CASE nIndex OF
	0: // idle state
		Inspect := 0;
	10: // trigger the camera
		IF GetCameraData() = 1 THEN
			Count := CameraData.Results.Count;
			CountStart := CameraData.Results.Count;
			nIndex := 11;
		END_IF
	11: // trigger camera
		Trigger := TRUE;
		nIndex := 12;
	12: // wait 250 ms
		CameraTON.IN := TRUE;
		IF CameraTON.Q THEN
			CameraTON.IN := FALSE;
			nIndex := 15;
		END_IF
		CameraTON();
	15: // wait for data to be updated
		CameraDataResult := GetCameraData();
		IF CameraDataResult = 1 THEN
			IF Count <> CameraData.Results.Count THEN
				CountFinish := CameraData.Results.Count;
				nIndex := 20;
				Trigger := FALSE;
			END_IF
		END_IF
	20: // Gather the data and analyze locations, etc.
		CameraDataResult := Compute(Execute := TRUE);
		IF CameraDataResult = 1 THEN	// could compute b/c found pattern
			Compute(Execute := FALSE);
			nIndex := 30;	
		ELSIF CameraDataResult = -1 THEN	// could not comput b/c no pattern found
			Compute(Execute := FALSE);
			nIndex := 50;
		END_IF
	30: // compute pass fail
		IF PassFail() THEN	// true = pass
			_pass := TRUE;
			_fail := FALSE;
			_noDetect := FALSE;
		ELSE
			_pass := FALSE;
			_fail := TRUE;
			_noDetect := FALSE;
		END_IF
		nIndex := 40;
	40: // done state
		Inspect := 1;
	50: // error state
		Inspect := -1;
		_noDetect := TRUE;		
		_pass := FALSE;
		_fail := FALSE;		
END_CASE
END_METHOD

METHOD MonitorParameters : BOOL
VAR_INPUT
END_VAR
IF angle <> _hmiParameters.angle THEN
	angle := _hmiParameters.angle;
END_IF

IF CalibrationDistance <> _hmiParameters.calibrationDistance THEN
	CalibrationDistance := _hmiParameters.calibrationDistance;
END_IF

IF pitchColumn <> _hmiParameters.pitchColumn THEN
	pitchColumn := _hmiParameters.pitchColumn;
END_IF

IF pitchRow <> _hmiParameters.pitchRow THEN
	pitchRow := _hmiParameters.pitchRow;
END_IF
END_METHOD

PROPERTY NoDetect : BOOL
GET
NoDetect := _noDetect;
END_GET
SET
_noDetect := NoDetect;
END_SET
END_PROPERTY

PROPERTY Parameters : ST_CameraParameters
GET
Parameters := _parameters;
END_GET
SET
_parameters := Parameters;
_hmiParameters := Parameters;
fbMessageLoaded.Send(0);
END_SET
END_PROPERTY

PROPERTY Pass : BOOL
GET
Pass := _pass;
END_GET
SET
_pass := Pass;
END_SET
END_PROPERTY

METHOD PassFail : BOOL
VAR_INPUT
END_VAR
PassFail := TRUE; // set to pass and overwrite if anything causes failure;

// cut length
IF _tubeParameters.AdjustmentLength + CutLength > _tubeParameters.MaxLength OR
	_tubeParameters.AdjustmentLength + CutLength < _tubeParameters.MinLength THEN
		PassFail := FALSE;
END_IF

// delta x
IF ABS(_tubeParameters.AdjustmentX + DeltaXmm) > _tubeParameters.ResultToleranceX THEN
	PassFail := FALSE;
END_IF

// delta y
IF ABS(_tubeParameters.AdjustmentY + DeltaYmm) > _tubeParameters.ResultToleranceY THEN
	PassFail := FALSE;
END_IF

// height
IF CutHeight < _tubeParameters.MinHeight OR CutHeight > _tubeParameters.MaxHeight THEN
	PassFail := FALSE;
END_IF
END_METHOD

PROPERTY PatternMatchX : LREAL
GET
PatternMatchX := REAL_TO_LREAL(CameraData.Results.PatternMatchColumn);
END_GET
END_PROPERTY

PROPERTY PatternMatchY : LREAL
GET
PatternMatchY := REAL_TO_LREAL(CameraData.Results.PatternMatchRow);
END_GET
END_PROPERTY

PROPERTY PatternX1 : LREAL
GET
PatternX1 := _patternX1;
END_GET
SET
_patternX1 := PatternX1;
END_SET
END_PROPERTY

PROPERTY PatternX2 : LREAL
GET
PatternX2 := _patternX2;
END_GET
SET
_patternX2 := PatternX2;
END_SET
END_PROPERTY

PROPERTY PatternX3 : LREAL
GET
PatternX3 := _patternX3;
END_GET
SET
_patternX3 := PatternX3;
END_SET
END_PROPERTY

PROPERTY PatternY1 : LREAL
GET
PatternY1 := _patternY1;
END_GET
SET
_patternY1 := PatternY1;
END_SET
END_PROPERTY

PROPERTY PatternY2 : LREAL
GET
PatternY2 := _patternY2;
END_GET
SET
_patternY2 := PatternY2;
END_SET
END_PROPERTY

PROPERTY PatternY3 : LREAL
GET
PatternY3 := _patternY3;
END_GET
SET
_patternY3 := PatternY3;
END_SET
END_PROPERTY

PROPERTY pitchColumn : LREAL
GET
pitchColumn := _parameters.pitchColumn;
END_GET
SET
fbMessageChange.ipArguments.Clear().AddString('pitchColumn').AddLReal(_parameters.pitchColumn).AddLReal(pitchColumn);
fbMessageChange.Send(0);
_parameters.pitchColumn := pitchColumn;
END_SET
END_PROPERTY

PROPERTY PitchMmToPixel : LREAL
GET
PitchMmToPixel := _hmiParameters.pitchRow;
END_GET
END_PROPERTY

PROPERTY pitchRow : LREAL
GET
pitchRow := _parameters.pitchRow;
END_GET
SET
fbMessageChange.ipArguments.Clear().AddString('pitchRow').AddLReal(_parameters.pitchRow).AddLReal(pitchRow);
fbMessageChange.Send(0);
_parameters.pitchRow := pitchRow;
END_SET
END_PROPERTY

METHOD SelectCameraProgram : INT
VAR_INPUT
	Execute	: BOOL;
END_VAR
VAR_INST
	fbMBRegWrite 	: FB_MBWriteRegs;	// for writing command, name; offset is 2000
	fbMBCoilWrite	: FB_MBWriteCoils;	// for writing vision control; offset is 0
	fbMBReadInputs 	: FB_MBReadInputs; 	// for reading vision status; offset is 0
	nIndex			: INT;
	rTrig			: R_TRIG;
	JobLoadByName 	: WORD := 16#4000;
	temp 			: UDINT := 0;
	info 			: BOOL;
	i 				: WORD;
	strJobName 		: STRING;
	Message			: STRING(255);
	ErrorId			: UDINT;
	nQuantity 		: WORD;
	cbLength 		: UDINT;	
	attempt			: INT;
	attempt2		: INT;	
END_VAR
VAR
END_VAR
rTrig(CLK := Execute);
IF rTrig.Q THEN
	nIndex := 10;
	Message := '';
	ErrorId := 0;
	Attempt := 0;
	Attempt2 := 0;
	fbMBCoilWrite(
		bExecute := FALSE,
		sIPAddr := GVL.CameraIpAddress,
		nTCPPort := 502,
		nUnitID := 16#FF);
	fbMBRegWrite(
		bExecute := FALSE,
		sIPAddr := GVL.CameraIpAddress,
		nTCPPort := 502,
		nUnitID := 16#FF);
	fbMBReadInputs(
		bExecute := FALSE,
		sIPAddr := GVL.CameraIpAddress,
		nTCPPort := 502,
		nUnitID := 16#FF);
END_IF

IF NOT Execute THEN
	nIndex := 0;
END_IF

CASE nIndex OF
	0: // idle state
		SelectCameraProgram := 0;
	10: // check if the program needs to change
		IF _previousTubeIndex = _tubeParameters.Index THEN
			nIndex := 75;
		ELSE
			nIndex := 15;
		END_IF
	15: // Reset everything to zero
		fbMBCoilWrite(
			nQuantity := 32,
			nMBAddr := 0,
			cbLength := 4,
			pSrcAddr := ADR(temp),
			bExecute := TRUE);
		IF NOT fbMBCoilWrite.bBusy THEN
			fbMBCoilWrite(bExecute := FALSE);
			nIndex := 20;
		END_IF
		IF fbMBCoilWrite.bError THEN
			Message := 'Error in state 15';
			ErrorId := fbMBCoilWrite.nErrId;
			fbMBCoilWrite(bExecute := FALSE);
			nIndex := 85;
		END_IF
	20: // place camera offline by setting the set offline bit high 
		// modbus coil offset is 0
		// byte 0, bit 7 is the bit for forcing the camera to be offline
		info := TRUE;
		fbMBCoilWrite(
			sIPAddr := GVL.CameraIpAddress,
			nTCPPort := 502,
			nUnitID := 16#FF,
			nQuantity := 1,
			nMBAddr := 7,
			cbLength := 1,
			pSrcAddr := ADR(Info),
			bExecute := TRUE);
		IF NOT fbMBCoilWrite.bBusy THEN
			fbMBCoilWrite(bExecute := FALSE);
			nIndex := 30;
			END_IF
		IF fbMBCoilWrite.bError THEN
			Message := 'Error in state 20';
			ErrorId := fbMBCoilWrite.nErrId;
			fbMBCoilWrite(bExecute := FALSE);
			nIndex := 85;
		END_IF		
	30: // write the job load by name command into Word 0 of the input block 
		// job load by name command is 0x4000
		// this goes into holding register start which is at 2000
		fbMBRegWrite(
			nQuantity := 1,
			nMBAddr := GVL.ModbusWriteOffset,
			cbLength := 2,
			pSrcAddr := ADR(JobLoadByName),
			bExecute := TRUE);
		IF NOT fbMBRegWrite.bBusy THEN
			fbMBRegWrite(bExecute := FALSE);
			attempt := attempt + 1;
			IF attempt > 2 THEN
				attempt := 0;
				nIndex := 40;
			END_IF
		END_IF
		IF fbMBRegWrite.bError THEN
			Message := 'Error in state 30';
			ErrorId := fbMBRegWrite.nErrId;
			fbMBRegWrite(bExecute := FALSE);
			nIndex := 85;

		END_IF
	40: // write the job name to Word 1 - 2000 (UserData).  Job name must be null terminated
		// a 0 must be in the byte immediately following the job name
		strJobName := CONCAT('SDCARD/Tube', INT_TO_STRING(_tubeParameters.Index));
		strJobName := CONCAT(strJobName, '.job');
		cbLength := 18; // INT_TO_UDINT(LEN(strJobName) + 1);
		nQuantity := 9; //REAL_TO_WORD(UDINT_TO_REAL(cbLength)/2);
		fbMBRegWrite(
			bExecute := TRUE,
			nQuantity := nQuantity,
			nMBAddr := GVL.ModbusWriteOffset + 1,
	//		nQuantity := nQuantity, // number of words
			cbLength := cbLength, // byte size
			pSrcAddr := ADR(strJobName));
		IF NOT fbMBRegWrite.bBusy THEN
			fbMBRegWrite(bExecute := FALSE);
			nIndex := 50;
		END_IF			
		IF fbMBRegWrite.bError THEN
			Message := 'Error in state 40';
			ErrorId := fbMBRegWrite.nErrId;
			fbMBRegWrite(bExecute := FALSE);
			Attempt2 := Attempt2 + 1;
			IF attempt2 > 2 THEN
				nIndex := 85;
			END_IF
		END_IF
		
	50: // Set the Execute Command bit in the vision control block
		//VisionControl.ExecuteCommand := TRUE;
		// Byte 0, bit 4 of vision control 
		info := TRUE;
		fbMBCoilWrite(
			nQuantity := 1,
			nMBAddr := 4,
			cbLength := 1,
			pSrcAddr := ADR(Info),
			bExecute := TRUE);
		IF NOT fbMBCoilWrite.bBusy THEN
			fbMBCoilWrite(bExecute := FALSE);
			nIndex := 60;
		END_IF
		IF fbMBCoilWrite.bError	THEN
			fbMBCoilWrite(bExecute := FALSE);
			nIndex := 85;
			Message := 'error in state 50';
			errorid := fbMBCoilWrite.nErrId;
		END_IF
	60: // wait for command complete of command failed to be set before clearing the execute
		// command bit and the offline bit
		fbMBReadInputs(
			sIPAddr := GVL.CameraIpAddress,
			nTCPPort := 502,
			nUnitID := 16#FF,
			nQuantity := 32,
			nMBAddr := 0,
			cbLength := 4,
			pDestAddr := ADR(VisionStatus),
			bExecute := TRUE);
		IF NOT fbMBReadInputs.bBusy THEN
			fbMBReadInputs(bExecute := FALSE);
			IF VisionStatus[1].6 OR VisionStatus[1].5 THEN
				nIndex := 70;
				IF VisionStatus[1].6 THEN
					nIndex := 80;
					Message := 'VisionSatus[1].6 is true.';
				END_IF
			END_IF
		END_IF
		IF fbMBReadInputs.bError THEN
			fbMBReadInputs(bExecute := FALSE);
			nIndex := 85;
			Errorid := fbMBReadInputs.nErrId;
			Message := 'errror in state 60.';
		END_IF
	70: // done state
		fbMBCoilWrite(
			nQuantity := 32,
			nMBAddr := 0,
			cbLength := 4,
			pSrcAddr := ADR(temp),
			bExecute := TRUE);
		IF NOT fbMBCoilWrite.bBusy THEN
			fbMBCoilWrite(bExecute := FALSE);
			nIndex := 75;
		END_IF
		IF fbMBCoilWrite.bError THEN
			fbMBCoilWrite(bExecute := FALSE);
			nIndex := 85;
			Message := 'error in state 70';
			ErrorID := fbMBCoilWrite.nErrId;			
		END_IF
	75: // done state
		_previousTubeIndex := _tubeParameters.Index;
		SelectCameraProgram := 1;
	80: // error state
		fbMBCoilWrite(
			nQuantity := 32,
			nMBAddr := 0,
			cbLength := 4,
			pSrcAddr := ADR(temp),
			bExecute := TRUE);
		IF NOT fbMBCoilWrite.bBusy THEN
			fbMBCoilWrite(bExecute := FALSE);
			nIndex := 85;
		END_IF

	85: // error state
		SelectCameraProgram := -1;
END_CASE





(*
SelectCameraProgram := 0;
fbMBRegWrite.bExecute := TRUE;

fbMBRegWrite.sIPAddr := GVL.CameraIpAddress;
fbMBRegWrite.nTCPPort := 502;
fbMBRegWrite.nUnitID := 16#FF;
fbMBRegWrite.nQuantity := 2; // words to write
fbMBRegWrite.nMBAddr := GVL.ModbusWriteOffset;
fbMBRegWrite.cbLength := SIZEOF(_tubeSelection);
fbMBRegWrite.pSrcAddr := ADR(_tubeSelection);

fbMBRegWrite();

IF NOT fbMBRegWrite.bBusy THEN
	IF NOT fbMBRegWrite.bError THEN
		fbMBRegWrite(bExecute := FALSE);
		SelectCameraProgram := 1;
	ELSE
		fbMBRegWrite(bExecute := FALSE);
		SelectCameraProgram := -1;		
	END_IF
END_IF
*)
END_METHOD

METHOD TriggerCamera : BOOL
VAR_INPUT
	Execute	: BOOL;
END_VAR
VAR_INST
	rTrig	: R_TRIG;
	nIndex	: INT;
	Counter	: REAL;
END_VAR
rTrig(CLK := Execute);
IF rTrig.Q THEN
	nIndex := 10;
	Trigger	:= FALSE;
END_IF

IF NOT Execute THEN
	nIndex := 0;
END_IF

CASE nIndex OF
	0: // idle state
		TriggerCamera := FALSE;
	10: // get the camera count
		IF GetCameraData() = 1 THEN
			Counter := CameraData.Results.Count;
			nIndex := 20;
		END_IF
	20: // trigger the camera	
		Trigger := TRUE;
		IF GetCameraData() = 1 THEN
			nIndex := 30;
		END_IF
	30: // updated?
		IF Counter <> CameraData.Results.Count THEN
			Trigger := FALSE;
			nIndex := 40;
		ELSE
			nIndex := 20;
		END_IF
	40: // done state
		TriggerCamera := TRUE;
END_CASE
END_METHOD

PROPERTY TubeParameters : ST_TubeParameters
GET
TubeParameters := _tubeParameters;
END_GET
SET
_tubeParameters := TubeParameters;
END_SET
END_PROPERTY

PROPERTY xEllipseCenter : LREAL
GET
xEllipseCenter := _xEllipseCenter;
END_GET
END_PROPERTY

PROPERTY yEllipseCenter : LREAL
GET
yEllipseCenter := _yEllipseCenter;
END_GET
END_PROPERTY

END_FUNCTION_BLOCK

// ---- Ellipse/FB_SecondOrder.TcPOU
FUNCTION_BLOCK FB_SecondOrder
VAR_INPUT
END_VAR
VAR_OUTPUT
END_VAR
VAR CONSTANT
	order : INT := 2;
END_VAR

METHOD Determinant2x2 : BOOL
VAR_INPUT
	ptrDeterminant	: POINTER TO LREAL;
	ptrMatrix		: POINTER TO ARRAY[1..2,1..2] OF LREAL;	
END_VAR
ptrDeterminant^ := ptrMatrix^[2,2]*ptrMatrix^[1,1] - ptrMatrix^[1,2]*ptrMatrix^[2,1];
END_METHOD

METHOD Determinant3x3 : BOOL
VAR_INPUT
	ptrDeterminant	: POINTER TO LREAL;
	ptrMatrix		: POINTER TO ARRAY[1..3,1..3] OF LREAL;
END_VAR
VAR
	Matrix3x3		: ARRAY[1..3,1..3] OF LREAL;
	Element1		: LREAL;
	Element2		: LREAL;
	RowMultiplier	: LREAL;
	i				: INT;
	j				: INT;
	row 			: INT;
	currentRow		: INT;
	temp			: LREAL;
	Swap			: BOOL;
	index			: INT;
	found			: BOOL;
END_VAR
Matrix3x3 := ptrMatrix^;
Swap := FALSE;
FOR index := 1 TO order DO
	IF Matrix3x3[index,index] = 0 THEN
		found := FALSE;
		FOR i:=index+1 TO 3 DO
			IF Matrix3x3[index,i] <> 0 THEN
				row := i;
				found := TRUE;
				EXIT;
			END_IF
		END_FOR
		// swap current row with found row
		IF found THEN
			FOR i := 1 TO order+1 DO
				temp := Matrix3x3[i,index];
				Matrix3x3[i,index] := Matrix3x3[i,row];
				Matrix3x3[i,row] := temp;
			END_FOR
			Swap := NOT Swap;
		ELSE
			ptrDeterminant^ := 0;
			Determinant3x3 := FALSE;
			RETURN;
		END_IF
	END_IF
	
	FOR j := index+1 TO order+1 DO
		Element1 := Matrix3x3[index,index];
		Element2 := Matrix3x3[index,j];
		IF Element2 <> 0 THEN
			RowMultiplier := Element2/Element1;
			FOR i := 1 TO order+1 DO
				Matrix3x3[i,j] := Matrix3x3[i,j] - RowMultiplier*Matrix3x3[i,index];
			END_FOR
		END_IF
	END_FOR
END_FOR

ptrDeterminant^ := 1;
FOR i := 1 TO order+1 DO
	ptrDeterminant^ := ptrDeterminant^ * Matrix3x3[i,i];
END_FOR

IF Swap THEN
	ptrDeterminant^ := ptrDeterminant^ * (-1);
END_IF	
Determinant3x3 := TRUE;
END_METHOD

METHOD Determinant4x4 : BOOL
VAR_INPUT
	ptrDeterminant	: POINTER TO LREAL;
	ptrMatrix		: POINTER TO ARRAY[1..4,1..4] OF LREAL;
END_VAR
VAR
	Matrix4x4		: ARRAY[1..4,1..4] OF LREAL;
	Element1		: LREAL;
	Element2		: LREAL;
	RowMultiplier	: LREAL;
	i				: INT;
	j				: INT;
	row 			: INT;
	currentRow		: INT;
	temp			: LREAL;
	Swap			: BOOL;
	index			: INT;
	found			: BOOL;
END_VAR
Matrix4x4 := ptrMatrix^;
Swap := FALSE;
FOR index := 1 TO 3 DO
	IF Matrix4x4[index,index] = 0 THEN
		found := FALSE;
		FOR i:=index+1 TO 4 DO
			IF Matrix4x4[index,i] <> 0 THEN
				row := i;
				found := TRUE;
				EXIT;
			END_IF
		END_FOR
		// swap current row with found row
		IF found THEN
			FOR i := 1 TO 4 DO
				temp := Matrix4x4[i,index];
				Matrix4x4[i,index] := Matrix4x4[i,row];
				Matrix4x4[i,row] := temp;
			END_FOR
			Swap := NOT Swap;
		ELSE
			ptrDeterminant^ := 0;
			Determinant4x4 := FALSE;
			RETURN;
		END_IF
	END_IF
	
	FOR j := index+1 TO 4 DO
		Element1 := Matrix4x4[index,index];
		Element2 := Matrix4x4[index,j];
		IF Element2 <> 0 THEN
			RowMultiplier := Element2/Element1;
			FOR i := 1 TO 4 DO
				Matrix4x4[i,j] := Matrix4x4[i,j] - RowMultiplier*Matrix4x4[i,index];
			END_FOR
		END_IF
	END_FOR
END_FOR

ptrDeterminant^ := 1;
FOR i := 1 TO 4 DO
	ptrDeterminant^ := ptrDeterminant^ * Matrix4x4[i,i];
END_FOR

IF Swap THEN
	ptrDeterminant^ := ptrDeterminant^ * (-1);
END_IF	
Determinant4x4 := TRUE;
END_METHOD

METHOD Determinant5x5 : BOOL
VAR_INPUT
	ptrDeterminant	: POINTER TO LREAL;
	ptrMatrix		: POINTER TO ARRAY[1..5,1..5] OF LREAL;
END_VAR
VAR
	Matrix5x5		: ARRAY[1..5,1..5] OF LREAL;
	Element1		: LREAL;
	Element2		: LREAL;
	RowMultiplier	: LREAL;
	i				: INT;
	j				: INT;
	row 			: INT;
	currentRow		: INT;
	temp			: LREAL;
	Swap			: BOOL;
	index			: INT;
	found			: BOOL;
END_VAR
Matrix5x5 := ptrMatrix^;
Swap := FALSE;
FOR index := 1 TO 4 DO
	IF Matrix5x5[index,index] = 0 THEN
		found := FALSE;
		FOR i:=index+1 TO 5 DO
			IF Matrix5x5[index,i] <> 0 THEN
				row := i;
				found := TRUE;
				EXIT;
			END_IF
		END_FOR
		// swap current row with found row
		IF found THEN
			FOR i := 1 TO 5 DO
				temp := Matrix5x5[i,index];
				Matrix5x5[i,index] := Matrix5x5[i,row];
				Matrix5x5[i,row] := temp;
			END_FOR
			Swap := NOT Swap;
		ELSE
			ptrDeterminant^ := 0;
			Determinant5x5 := FALSE;
			RETURN;
		END_IF
	END_IF
	
	FOR j := index+1 TO 5 DO
		Element1 := Matrix5x5[index,index];
		Element2 := Matrix5x5[index,j];
		IF Element2 <> 0 THEN
			RowMultiplier := Element2/Element1;
			FOR i := 1 TO 5 DO
				Matrix5x5[i,j] := Matrix5x5[i,j] - RowMultiplier*Matrix5x5[i,index];
			END_FOR
		END_IF
	END_FOR
END_FOR

ptrDeterminant^ := 1;
FOR i := 1 TO 5 DO
	ptrDeterminant^ := ptrDeterminant^ * Matrix5x5[i,i];
END_FOR

IF Swap THEN
	ptrDeterminant^ := ptrDeterminant^ * (-1);
END_IF	
Determinant5x5 := TRUE;
END_METHOD

METHOD FindCoefficients : BOOL
VAR_INPUT
	xValues		: POINTER TO ARRAY[1..GVL.NumberVisionPoints] OF LREAL;
	yValues		: POINTER TO ARRAY[1..GVL.NumberVisionPoints] OF LREAL;
	Coefficients: POINTER TO ARRAY[1..3] OF LREAL;
END_VAR
VAR_INST 
	xMatrix		: ARRAY[1..3, 1..GVL.NumberVisionPoints] OF LREAL;
	xTMatrix	: ARRAY[1..GVL.NumberVisionPoints, 1..3] OF LREAL; 
	xTxMatrix	: ARRAY[1..3,1..3] OF LREAL;
	xTxInverse	: ARRAY[1..3,1..3] OF LREAL;
	xTyMatrix	: ARRAY[1..3] OF LREAL;
	i			: INT;
	j			: INT;
	k			: INT;
	DotProduct	: LREAL;
END_VAR
// fill out x matrix
// fill out transpose of x matrix
FOR i := 1 TO order+1 DO	// column
	FOR j := 1 TO GVL.NumberVisionPoints DO
		xMatrix[i,j] := EXPT((xValues^[j]),(i-1));	
		xTMatrix[j,i] := xMatrix[i,j];
	END_FOR
END_FOR

// fill out xT * x 
FOR i := 1 TO order+1 DO		// rows
	FOR j := 1 TO order+1 DO	
		DotProduct := 0;
		FOR k := 1 TO GVL.NumberVisionPoints DO
			DotProduct := DotProduct + xTMatrix[k,i]*xMatrix[j,k];
		END_FOR
		xTxMatrix[j,i] := DotProduct;
	END_FOR
END_FOR

// find out the inverse of xT*x
Inverse(ptrMatrix := ADR(xTxMatrix), ptrInverse := ADR(xTxInverse));

// multiple xT*y
FOR i := 1 TO order+1 DO 
	DotProduct := 0;
	FOR j := 1 TO GVL.NumberVisionPoints DO
		DotProduct := DotProduct + xTMatrix[j,i] * yValues^[j];
	END_FOR
	xTyMatrix[i] := DotProduct;
END_FOR

// multiply xTxInverse by xTy
FOR i := 1 TO order+1 DO
	DotProduct := 0;
	FOR j := 1 TO order+1 DO
		DotProduct := DotProduct + xTxInverse[j,i]*xTyMatrix[j];
	END_FOR
	Coefficients^[i] := DotProduct;
END_FOR
END_METHOD

METHOD FindPeak : LREAL
VAR_INPUT
	xValues		: POINTER TO ARRAY[1..GVL.NumberVisionPoints] OF LREAL;
	yValues		: POINTER TO ARRAY[1..GVL.NumberVisionPoints] OF LREAL;
	xPeak		: POINTER TO LREAL;
END_VAR
VAR
	Coefficients: ARRAY[1..3] OF LREAL;	
	a			: LREAL;
	b			: LREAL;
END_VAR
FindCoefficients(xValues := xValues, yValues := yValues, Coefficients := ADR(Coefficients));
a := Coefficients[3];
b := Coefficients[2];
xPeak^ := -b/(2*a);
END_METHOD

METHOD Inverse : BOOL
VAR_INPUT
	ptrMatrix		: POINTER TO ARRAY[1..3,1..3] OF LREAL;
	ptrInverse		: POINTER TO ARRAY[1..3,1..3] OF LREAL;
END_VAR
VAR_INST
	Matrix3x3		: ARRAY[1..3,1..3] OF LREAL;
	Determinant		: LREAL;
	Matrix			: ARRAY[1..3,1..3] OF LREAL; // matrix of minors
	Matrix2x2		: ARRAY[1..2,1..2] OF LREAL;
	_Cofactor		: LREAL;
	i				: INT;
	j				: INT;
	SignRow			: BOOL;
	SignColumn		: BOOL;
END_VAR
Matrix3x3 := ptrMatrix^;

IF Determinant3x3(ptrDeterminant := ADR(Determinant), ptrMatrix := ptrMatrix) THEN
	Determinant := 1 / Determinant;

	// matrix of minors
	// column 1:
	Matrix2x2[1,1] := Matrix3x3[2,2];
	Matrix2x2[1,2] := Matrix3x3[2,3];
	Matrix2x2[2,1] := Matrix3x3[3,2];
	Matrix2x2[2,2] := Matrix3x3[3,3];
	Determinant2x2(ADR(Matrix[1,1]), ADR(Matrix2x2));

	Matrix2x2[1,1] := Matrix3x3[2,1];
	Matrix2x2[1,2] := Matrix3x3[2,3];
	Matrix2x2[2,1] := Matrix3x3[3,1];
	Matrix2x2[2,2] := Matrix3x3[3,3];
	Determinant2x2(ADR(Matrix[1,2]), ADR(Matrix2x2));

	Matrix2x2[1,1] := Matrix3x3[2,1];
	Matrix2x2[1,2] := Matrix3x3[2,2];
	Matrix2x2[2,1] := Matrix3x3[3,1];
	Matrix2x2[2,2] := Matrix3x3[3,2];
	Determinant2x2(ADR(Matrix[1,3]), ADR(Matrix2x2));
	
	// column 2:
	Matrix2x2[1,1] := Matrix3x3[1,2];
	Matrix2x2[1,2] := Matrix3x3[1,3];
	Matrix2x2[2,1] := Matrix3x3[3,2];
	Matrix2x2[2,2] := Matrix3x3[3,3];
	Determinant2x2(ADR(Matrix[2,1]), ADR(Matrix2x2));

	Matrix2x2[1,1] := Matrix3x3[1,1];
	Matrix2x2[1,2] := Matrix3x3[1,3];
	Matrix2x2[2,1] := Matrix3x3[3,1];
	Matrix2x2[2,2] := Matrix3x3[3,3];
	Determinant2x2(ADR(Matrix[2,2]), ADR(Matrix2x2));

	Matrix2x2[1,1] := Matrix3x3[1,1];
	Matrix2x2[1,2] := Matrix3x3[1,2];
	Matrix2x2[2,1] := Matrix3x3[3,1];
	Matrix2x2[2,2] := Matrix3x3[3,2];
	Determinant2x2(ADR(Matrix[2,3]), ADR(Matrix2x2));

	// column 3:
	Matrix2x2[1,1] := Matrix3x3[1,2];
	Matrix2x2[1,2] := Matrix3x3[1,3];
	Matrix2x2[2,1] := Matrix3x3[2,2];
	Matrix2x2[2,2] := Matrix3x3[2,3];
	Determinant2x2(ADR(Matrix[3,1]), ADR(Matrix2x2));

	Matrix2x2[1,1] := Matrix3x3[1,1];
	Matrix2x2[1,2] := Matrix3x3[1,3];
	Matrix2x2[2,1] := Matrix3x3[2,1];
	Matrix2x2[2,2] := Matrix3x3[2,3];
	Determinant2x2(ADR(Matrix[3,2]), ADR(Matrix2x2));

	Matrix2x2[1,1] := Matrix3x3[1,1];
	Matrix2x2[1,2] := Matrix3x3[1,2];
	Matrix2x2[2,1] := Matrix3x3[2,1];
	Matrix2x2[2,2] := Matrix3x3[2,2];
	Determinant2x2(ADR(Matrix[3,3]), ADR(Matrix2x2));
	
	// switch the signs	
	SignRow := TRUE;
	SignColumn := TRUE;
	FOR i := 1 TO order+1 DO
		FOR j := 1 TO order+1 DO
			IF NOT SignRow THEN
				Matrix[i,j] := (-1) * Matrix[i,j];
			END_IF
			SignRow := NOT SignRow;
		END_FOR
		SignColumn := NOT SignColumn;
		SignRow := SignColumn;
	END_FOR
	// transpose 
	Transpose(ADR(Matrix),ptrInverse);
	FOR i := 1 TO order+1 DO
		FOR j := 1 TO order+1 DO
			ptrInverse^[i,j] := Determinant * ptrInverse^[i,j];
		END_FOR
	END_FOR
	
	Inverse := TRUE;
ELSE
	Inverse := FALSE;
END_IF
END_METHOD

METHOD Transpose : BOOL
VAR_INPUT
	ptrMatrix		: POINTER TO ARRAY[1..3,1..3] OF LREAL;
	ptrTranspose	: POINTER TO ARRAY[1..3,1..3] OF LREAL;
END_VAR
VAR
	i				: INT;
	j				: INT;
END_VAR
FOR i := 1 TO order+1 DO
	FOR j := 1 TO order+1 DO
		ptrTranspose^[j,i] := ptrMatrix^[i,j];
	END_FOR
END_FOR
END_METHOD

END_FUNCTION_BLOCK

// ---- Ellipse/FB_FourthOrder.TcPOU
FUNCTION_BLOCK FB_FourthOrder
VAR_INPUT
END_VAR
VAR_OUTPUT
END_VAR
VAR CONSTANT
	order : INT := 4;
END_VAR

METHOD Cofactor : BOOL
VAR_INPUT
	ptrMatrix5x5	: POINTER TO ARRAY[1..5,1..5] OF LREAL;
	ptrCofactor		: POINTER TO LREAL;
	row				: INT;
	column			: INT;
END_VAR
VAR
	Matrix4x4	: ARRAY[1..4,1..4] OF LREAL;	
	i			: INT;
	j			: INT;
	k			: INT;
	m			: INT;
END_VAR
k := 1;
FOR i := 1 TO order+1 DO				// columns
	m := 1;
	IF i <> column THEN						
		FOR j := 1 TO order+1 DO		
			IF j <> row THEN
				Matrix4x4[k,m] := ptrMatrix5x5^[i,j];
				m := m + 1;
			END_IF
		END_FOR
		k := k + 1;
	END_IF
END_FOR

IF Determinant4x4(ptrDeterminant := ptrCofactor, ptrMatrix := ADR(Matrix4x4)) THEN
	Cofactor := TRUE;
ELSE
	Cofactor := FALSE;
END_IF
END_METHOD

METHOD Determinant4x4 : BOOL
VAR_INPUT
	ptrDeterminant	: POINTER TO LREAL;
	ptrMatrix		: POINTER TO ARRAY[1..4,1..4] OF LREAL;
END_VAR
VAR
	Matrix4x4		: ARRAY[1..4,1..4] OF LREAL;
	Element1		: LREAL;
	Element2		: LREAL;
	RowMultiplier	: LREAL;
	i				: INT;
	j				: INT;
	row 			: INT;
	currentRow		: INT;
	temp			: LREAL;
	Swap			: BOOL;
	index			: INT;
	found			: BOOL;
END_VAR
Matrix4x4 := ptrMatrix^;
Swap := FALSE;
FOR index := 1 TO 3 DO
	IF Matrix4x4[index,index] = 0 THEN
		found := FALSE;
		FOR i:=index+1 TO 4 DO
			IF Matrix4x4[index,i] <> 0 THEN
				row := i;
				found := TRUE;
				EXIT;
			END_IF
		END_FOR
		// swap current row with found row
		IF found THEN
			FOR i := 1 TO 4 DO
				temp := Matrix4x4[i,index];
				Matrix4x4[i,index] := Matrix4x4[i,row];
				Matrix4x4[i,row] := temp;
			END_FOR
			Swap := NOT Swap;
		ELSE
			ptrDeterminant^ := 0;
			Determinant4x4 := FALSE;
			RETURN;
		END_IF
	END_IF
	
	FOR j := index+1 TO 4 DO
		Element1 := Matrix4x4[index,index];
		Element2 := Matrix4x4[index,j];
		IF Element2 <> 0 THEN
			RowMultiplier := Element2/Element1;
			FOR i := 1 TO 4 DO
				Matrix4x4[i,j] := Matrix4x4[i,j] - RowMultiplier*Matrix4x4[i,index];
			END_FOR
		END_IF
	END_FOR
END_FOR

ptrDeterminant^ := 1;
FOR i := 1 TO 4 DO
	ptrDeterminant^ := ptrDeterminant^ * Matrix4x4[i,i];
END_FOR

IF Swap THEN
	ptrDeterminant^ := ptrDeterminant^ * (-1);
END_IF	
Determinant4x4 := TRUE;
END_METHOD

METHOD Determinant5x5 : BOOL
VAR_INPUT
	ptrDeterminant	: POINTER TO LREAL;
	ptrMatrix		: POINTER TO ARRAY[1..5,1..5] OF LREAL;
END_VAR
VAR
	Matrix5x5		: ARRAY[1..5,1..5] OF LREAL;
	Element1		: LREAL;
	Element2		: LREAL;
	RowMultiplier	: LREAL;
	i				: INT;
	j				: INT;
	row 			: INT;
	currentRow		: INT;
	temp			: LREAL;
	Swap			: BOOL;
	index			: INT;
	found			: BOOL;
END_VAR
Matrix5x5 := ptrMatrix^;
Swap := FALSE;
FOR index := 1 TO 4 DO
	IF Matrix5x5[index,index] = 0 THEN
		found := FALSE;
		FOR i:=index+1 TO 5 DO
			IF Matrix5x5[index,i] <> 0 THEN
				row := i;
				found := TRUE;
				EXIT;
			END_IF
		END_FOR
		// swap current row with found row
		IF found THEN
			FOR i := 1 TO 5 DO
				temp := Matrix5x5[i,index];
				Matrix5x5[i,index] := Matrix5x5[i,row];
				Matrix5x5[i,row] := temp;
			END_FOR
			Swap := NOT Swap;
		ELSE
			ptrDeterminant^ := 0;
			Determinant5x5 := FALSE;
			RETURN;
		END_IF
	END_IF
	
	FOR j := index+1 TO 5 DO
		Element1 := Matrix5x5[index,index];
		Element2 := Matrix5x5[index,j];
		IF Element2 <> 0 THEN
			RowMultiplier := Element2/Element1;
			FOR i := 1 TO 5 DO
				Matrix5x5[i,j] := Matrix5x5[i,j] - RowMultiplier*Matrix5x5[i,index];
			END_FOR
		END_IF
	END_FOR
END_FOR

ptrDeterminant^ := 1;
FOR i := 1 TO 5 DO
	ptrDeterminant^ := ptrDeterminant^ * Matrix5x5[i,i];
END_FOR

IF Swap THEN
	ptrDeterminant^ := ptrDeterminant^ * (-1);
END_IF	
Determinant5x5 := TRUE;
END_METHOD

METHOD FindCoefficients : BOOL
VAR_INPUT
	xValues		: POINTER TO ARRAY[1..GVL.NumberVisionPoints] OF LREAL;
	yValues		: POINTER TO ARRAY[1..GVL.NumberVisionPoints] OF LREAL;
	Coefficients: POINTER TO ARRAY[1..5] OF LREAL;
END_VAR
VAR_INST 
	xMatrix		: ARRAY[1..5, 1..GVL.NumberVisionPoints] OF LREAL;
	xTMatrix	: ARRAY[1..GVL.NumberVisionPoints, 1..5] OF LREAL; 
	xTxMatrix	: ARRAY[1..5,1..5] OF LREAL;
	xTxInverse	: ARRAY[1..5,1..5] OF LREAL;
	xTxXMatrix	: ARRAY[1..GVL.NumberVisionPoints,1..5] OF LREAL;
	xTyMatrix	: ARRAY[1..5] OF LREAL;
	i			: INT;
	j			: INT;
	k			: INT;
	DotProduct	: LREAL;
END_VAR
// fill out x matrix
// fill out transpose of x matrix
FOR i := 1 TO order+1 DO	// column
	FOR j := 1 TO GVL.NumberVisionPoints DO
		xMatrix[i,j] := EXPT((xValues^[j]),(i-1));	// column, row
		xTMatrix[j,i] := xMatrix[i,j];
	END_FOR
END_FOR

// fill out xT * x 
FOR i := 1 TO order+1 DO		// rows
	FOR j := 1 TO order+1 DO	
		DotProduct := 0;
		FOR k := 1 TO GVL.NumberVisionPoints DO
			DotProduct := DotProduct + xTMatrix[k,i]*xMatrix[j,k];
		END_FOR
		xTxMatrix[j,i] := DotProduct;
	END_FOR
END_FOR

// find out the inverse of xT*x
Inverse(ADR(xTxMatrix), ADR(xTxInverse));

// multiple xT*y
FOR i := 1 TO order+1 DO
	DotProduct := 0;
	FOR j := 1 TO GVL.NumberVisionPoints DO
		DotProduct := DotProduct + xTMatrix[j,i] * yValues^[j];
	END_FOR
	xTyMatrix[i] := DotProduct;
END_FOR

// multiply xTxInverse by xTy
FOR i := 1 TO order+1 DO
	DotProduct := 0;
	FOR j := 1 TO order+1 DO
		DotProduct := DotProduct + xTxInverse[j,i]*xTyMatrix[j];
	END_FOR
	Coefficients^[i] := DotProduct;
END_FOR
END_METHOD

METHOD FindYatX : BOOL
VAR_INPUT
	xValues			: POINTER TO ARRAY[1..GVL.NumberVisionPoints] OF LREAL;
	yValues			: POINTER TO ARRAY[1..GVL.NumberVisionPoints] OF LREAL;
	xPeak			: POINTER TO LREAL;
	yPeak			: POINTER TO LREAL;
END_VAR
VAR
	Coefficients	: ARRAY[1..5] OF LREAL;
END_VAR
FindCoefficients(xValues := xValues, yValues := yValues, Coefficients := ADR(Coefficients));
yPeak^ := Coefficients[1] + Coefficients[2] * xPeak^ + Coefficients[3]*EXPT(xPeak^,2) + 
		Coefficients[4]*EXPT(xPeak^,3) + Coefficients[5]*EXPT(xPeak^,4);
END_METHOD

METHOD Inverse : BOOL
VAR_INPUT
	ptrMatrix		: POINTER TO ARRAY[1..5,1..5] OF LREAL;
	ptrInverse		: POINTER TO ARRAY[1..5,1..5] OF LREAL;
END_VAR
VAR
	Determinant		: LREAL;
	Matrix			: ARRAY[1..5,1..5] OF LREAL;
	_Cofactor		: LREAL;
	i				: INT;
	j				: INT;
	SignRow: BOOL;
	SignColumn: BOOL;
END_VAR
IF Determinant5x5(ptrDeterminant := ADR(Determinant), ptrMatrix := ptrMatrix) THEN
	Determinant := 1 / Determinant;
	// get cofactors
	FOR i := 1 TO order+1 DO
		FOR j := 1 TO order+1 DO
			IF Cofactor(ptrMatrix5x5 := ptrMatrix, ptrCofactor := ADR(_Cofactor), row := i, column := j) THEN
				Matrix[i,j] := _Cofactor;
			ELSE
				Inverse := FALSE;
				RETURN;
			END_IF
		END_FOR
	END_FOR
	
	SignRow := TRUE;
	SignColumn := TRUE;
	FOR i := 1 TO order+1 DO
		FOR j := 1 TO order+1 DO
			IF NOT SignRow THEN
				Matrix[i,j] := (-1) * Matrix[i,j];
			END_IF
			SignRow := NOT SignRow;
		END_FOR
		SignColumn := NOT SignColumn;
		SignRow := SignColumn;
	END_FOR
	// transpose 
	Transpose(ADR(Matrix),ptrInverse);
	FOR i := 1 TO order+1 DO
		FOR j := 1 TO order+1 DO
			ptrInverse^[i,j] := Determinant * ptrInverse^[i,j];
		END_FOR
	END_FOR
	
	Inverse := TRUE;
ELSE
	Inverse := FALSE;
END_IF
END_METHOD

METHOD Transpose : BOOL
VAR_INPUT
	ptrMatrix		: POINTER TO ARRAY[1..5,1..5] OF LREAL;
	ptrTranspose	: POINTER TO ARRAY[1..5,1..5] OF LREAL;
END_VAR
VAR
	i				: INT;
	j				: INT;
END_VAR
FOR i := 1 TO order+1 DO
	FOR j := 1 TO order+1 DO
		ptrTranspose^[j,i] := ptrMatrix^[i,j];
	END_FOR
END_FOR
END_METHOD

END_FUNCTION_BLOCK

// ---- Ellipse/FB_Ellipse.TcPOU
FUNCTION_BLOCK FB_Ellipse
VAR_INPUT
END_VAR
VAR_OUTPUT
END_VAR
VAR CONSTANT
END_VAR
VAR
	_xValues				: ARRAY[1..GVL.NumberEllipsePoints] OF LREAL := [0,1,2,3,4,5,6,7,8,9];
	_yValues				: ARRAY[1..GVL.NumberEllipsePoints] OF LREAL := [5,4.975,4.899,4.770,4.583,4.330,4.000,3.571,3.000,2.179];

	m_residuals		: ARRAY[1..GVL.NumberEllipsePoints] OF LREAL;						// [NumDataPts x 1]
	m_design		: ARRAY[1..GVL.Unknowns, 1..GVL.NumberEllipsePoints] OF LREAL;		// [NumDataPts x 5]
	m_l				: ARRAY[1..GVL.NumberEllipsePoints] OF LREAL;						// [NumDataPts x 1]
	m_qweight		: ARRAY[1..GVL.NumberEllipsePoints, 1..GVL.NumberEllipsePoints] OF LREAL;	// [NumDataPts x NumDataPts]
	m_observations	: ARRAY[1..2,1..GVL.NumberEllipsePoints] OF LREAL; 				// [NumDataPts x 2]
	m_b				: ARRAY[1..2*GVL.NumberEllipsePoints, 1..GVL.NumberEllipsePoints] OF LREAL;	// [NumDataPts x NumDataPts*2]
	m_miny			: LREAL;
	m_maxy			: LREAL;
	m_minx			: LREAL;
	m_maxx			: LREAL;
	m_provisionals	: ARRAY[1..GVL.Unknowns] OF LREAL; // [5 x 1]
	m_solutions		: ARRAY[1..GVL.Unknowns] OF LREAL; // [5 x 1]

// junk
	_pa				: ARRAY[1..GVL.Unknowns, 1..GVL.NumberEllipsePoints] OF LREAL;	
	_atpa			: ARRAY[1..GVL.Unknowns, 1..GVL.Unknowns] OF LREAL;
	_atpaInverse		: ARRAY[1..GVL.Unknowns, 1..GVL.Unknowns] OF LREAL;
	_pl				: ARRAY[1..GVL.NumberEllipsePoints] OF LREAL; 
	_atpl			: ARRAY[1..GVL.Unknowns] OF LREAL;
	_cofactorMatrix	: ARRAY[1..5,1..5] OF LREAL;
	_cofactorMatrixSigned : ARRAY[1..5,1..5] OF LREAL;
	_cofactorMatrixT : ARRAY[1..5,1..5] OF LREAL;

END_VAR

METHOD AddObservation : BOOL
VAR_INPUT
END_VAR
VAR
	i	: INT;
END_VAR
m_minx := _xValues[1];
m_maxx := _xValues[1];
m_miny := _yValues[1];
m_maxy := _yValues[1];
FOR i := 1 TO GVL.NumberEllipsePoints DO
	m_observations[1,i] := _xValues[i];
	m_observations[2,i] := _yValues[i];
	IF _xValues[i] > m_maxx THEN
		m_maxx := _xValues[i];
	END_IF
	IF _xValues[i] < m_minx THEN
		m_minx := _xValues[i];
	END_IF
	IF _yValues[i] > m_maxy THEN
		m_maxy := _yValues[i];
	END_IF
	IF _yValues[i] < m_miny THEN
		m_miny := _yValues[i];
	END_IF
END_FOR
END_METHOD

PROPERTY centrex : LREAL
GET
centrex := m_provisionals[1];

(*
m_provisionals[1] := _centrex;
m_provisionals[2] := _centrey;
m_provisionals[3] := _major;
m_provisionals[4] := _minor;
m_provisionals[5] := _rotation;
*)
END_GET
END_PROPERTY

PROPERTY centrey : LREAL
GET
centrey := m_provisionals[2];

(*
m_provisionals[1] := _centrex;
m_provisionals[2] := _centrey;
m_provisionals[3] := _major;
m_provisionals[4] := _minor;
m_provisionals[5] := _rotation;
*)
END_GET
END_PROPERTY

METHOD Cofactor : BOOL
VAR_INPUT
	ptrMatrix5x5	: POINTER TO ARRAY[1..5,1..5] OF LREAL;
	ptrCofactor		: POINTER TO LREAL;
	row				: INT;
	column			: INT;
END_VAR
VAR
	Matrix4x4	: ARRAY[1..4,1..4] OF LREAL;	
	i			: INT;
	j			: INT;
	k			: INT;
	m			: INT;
END_VAR
k := 1;
FOR i := 1 TO 5 DO				// columns
	m := 1;
	IF i <> column THEN						
		FOR j := 1 TO 5 DO		
			IF j <> row THEN
				Matrix4x4[k,m] := ptrMatrix5x5^[i,j];
				m := m + 1;
			END_IF
		END_FOR
		k := k + 1;
	END_IF
END_FOR

IF Determinant4x4(ptrDeterminant := ptrCofactor, ptrMatrix := ADR(Matrix4x4)) THEN
	Cofactor := TRUE;
ELSE
	Cofactor := FALSE;
END_IF
END_METHOD

METHOD Compute : BOOL
VAR_INPUT
END_VAR
VAR_INST
	successful	: BOOL;
	iteration	: INT;
	bHasConverged	: BOOL;
	bIsDegenerate	: BOOL;
END_VAR
GenerateProvisionals();

successful := TRUE;
bHasConverged := FALSE;
bIsDegenerate := FALSE;

iteration := 0;

WHILE (TRUE) DO
	FormulateMatrices();
	IF (EvaluateUnknowns()) THEN
		iteration := iteration + 1;
		EvaluateAdjustedUnknowns();
		IF HasConverged() THEN
			bHasConverged := TRUE;
			EXIT;
		END_IF
		IF IsDegenerate(iteration) THEN
			bIsDegenerate := TRUE;
			EXIT;
		END_IF
	ELSE
		successful := FALSE;
		EXIT;
	END_IF	
END_WHILE

successful := successful AND (iteration > 0 AND iteration < GVL.MaxIterations);
IF successful THEN
	NormalizeAdjustedUnknowns();
	EvaluateResiduals();
//	EvaluateAdjustedObservations();
//	GlobalCheck();
//	ErrorAnalysis(iteration);
END_IF

Compute := successful;
END_METHOD

METHOD Determinant4x4 : BOOL
VAR_INPUT
	ptrDeterminant	: POINTER TO LREAL;
	ptrMatrix		: POINTER TO ARRAY[1..4,1..4] OF LREAL;
END_VAR
VAR
	Matrix4x4		: ARRAY[1..4,1..4] OF LREAL;
	Element1		: LREAL;
	Element2		: LREAL;
	RowMultiplier	: LREAL;
	i				: INT;
	j				: INT;
	row 			: INT;
	currentRow		: INT;
	temp			: LREAL;
	Swap			: BOOL;
	index			: INT;
	found			: BOOL;
END_VAR
Matrix4x4 := ptrMatrix^;
Swap := FALSE;
FOR index := 1 TO 3 DO
	IF Matrix4x4[index,index] = 0 THEN
		found := FALSE;
		FOR i:=index+1 TO 4 DO
			IF Matrix4x4[index,i] <> 0 THEN
				row := i;
				found := TRUE;
				EXIT;
			END_IF
		END_FOR
		// swap current row with found row
		IF found THEN
			FOR i := 1 TO 4 DO
				temp := Matrix4x4[i,index];
				Matrix4x4[i,index] := Matrix4x4[i,row];
				Matrix4x4[i,row] := temp;
			END_FOR
			Swap := NOT Swap;
		ELSE
			ptrDeterminant^ := 0;
			Determinant4x4 := FALSE;
			RETURN;
		END_IF
	END_IF
	
	FOR j := index+1 TO 4 DO
		Element1 := Matrix4x4[index,index];
		Element2 := Matrix4x4[index,j];
		IF Element2 <> 0 THEN
			RowMultiplier := Element2/Element1;
			FOR i := 1 TO 4 DO
				Matrix4x4[i,j] := Matrix4x4[i,j] - RowMultiplier*Matrix4x4[i,index];
			END_FOR
		END_IF
	END_FOR
END_FOR

ptrDeterminant^ := 1;
FOR i := 1 TO 4 DO
	ptrDeterminant^ := ptrDeterminant^ * Matrix4x4[i,i];
END_FOR

IF Swap THEN
	ptrDeterminant^ := ptrDeterminant^ * (-1);
END_IF	
Determinant4x4 := TRUE;
END_METHOD

METHOD Determinant5x5 : BOOL
VAR_INPUT
	ptrDeterminant	: POINTER TO LREAL;
	ptrMatrix		: POINTER TO ARRAY[1..5,1..5] OF LREAL;
END_VAR
VAR
	Matrix5x5		: ARRAY[1..5,1..5] OF LREAL;
	Element1		: LREAL;
	Element2		: LREAL;
	RowMultiplier	: LREAL;
	i				: INT;
	j				: INT;
	row 			: INT;
	currentRow		: INT;
	temp			: LREAL;
	Swap			: BOOL;
	index			: INT;
	found			: BOOL;
END_VAR
Matrix5x5 := ptrMatrix^;
Swap := FALSE;
FOR index := 1 TO 4 DO
	IF Matrix5x5[index,index] = 0 THEN
		found := FALSE;
		FOR i:=index+1 TO 5 DO
			IF Matrix5x5[index,i] <> 0 THEN
				row := i;
				found := TRUE;
				EXIT;
			END_IF
		END_FOR
		// swap current row with found row
		IF found THEN
			FOR i := 1 TO 5 DO
				temp := Matrix5x5[i,index];
				Matrix5x5[i,index] := Matrix5x5[i,row];
				Matrix5x5[i,row] := temp;
			END_FOR
			Swap := NOT Swap;
		ELSE
			ptrDeterminant^ := 0;
			Determinant5x5 := FALSE;
			RETURN;
		END_IF
	END_IF
	
	FOR j := index+1 TO 5 DO
		Element1 := Matrix5x5[index,index];
		Element2 := Matrix5x5[index,j];
		IF Element2 <> 0 THEN
			RowMultiplier := Element2/Element1;
			FOR i := 1 TO 5 DO
				Matrix5x5[i,j] := Matrix5x5[i,j] - RowMultiplier*Matrix5x5[i,index];
			END_FOR
		END_IF
	END_FOR
END_FOR

ptrDeterminant^ := 1;
FOR i := 1 TO 5 DO
	ptrDeterminant^ := ptrDeterminant^ * Matrix5x5[i,i];
END_FOR

IF Swap THEN
	ptrDeterminant^ := ptrDeterminant^ * (-1);
END_IF	
Determinant5x5 := TRUE;
END_METHOD

METHOD EllipseFit : BOOL
VAR_INPUT
	xValues	: ARRAY[1..GVL.NumberEllipsePoints] OF LREAL;
	yValues	: ARRAY[1..GVL.NumberEllipsePoints] OF LREAL;
END_VAR
VAR 
	i		: INT;
	x		: LREAL;
	y		: LREAL;
END_VAR
_xValues := xValues;
_yValues := yValues;
AddObservation();
Compute();
END_METHOD

METHOD ErrorAnalysis : BOOL
VAR_INPUT
	iteration	: INT;
END_VAR
END_METHOD

METHOD EvaluateAdjustedUnknowns : BOOL
VAR_INPUT
END_VAR
VAR
	i		: INT;
END_VAR
FOR i:=1 TO GVL.Unknowns DO
	m_provisionals[i] := m_provisionals[i] + m_solutions[i];
END_FOR
END_METHOD

METHOD EvaluateResiduals : BOOL
VAR
	i			: INT;
	j			: INT;
	k			: INT;
	DotProduct	: LREAL;
END_VAR
// m_residuals = prod(m_design, m_solution) - m_l

FOR i := 1 TO GVL.NumberEllipsePoints DO // rows
	DotProduct := 0;
	FOR j := 1 TO GVL.Unknowns DO
		DotProduct := DotProduct + m_design[j,i]*m_solutions[j];
	END_FOR
	m_residuals[i] := DotProduct;
END_FOR

FOR i := 1 TO GVL.NumberEllipsePoints DO
	m_residuals[i] := m_residuals[i] - m_l[i];
END_FOR
END_METHOD

METHOD EvaluateUnknowns : BOOL
VAR_INPUT
END_VAR
VAR
	pa				: ARRAY[1..GVL.Unknowns, 1..GVL.NumberEllipsePoints] OF LREAL;	
	atpa			: ARRAY[1..GVL.Unknowns, 1..GVL.Unknowns] OF LREAL;
	atpaInverse		: ARRAY[1..GVL.Unknowns, 1..GVL.Unknowns] OF LREAL;
	pl				: ARRAY[1..GVL.NumberEllipsePoints] OF LREAL; 
	atpl			: ARRAY[1..GVL.Unknowns] OF LREAL;
	i				: INT;
	j				: INT;
	k				: INT;
	DotProduct		: LREAL;
END_VAR
(*
1. pa := prod(m_qweight, m_design)
2. atpa := prod(trans(m_design), pa)
3. create a matrix variable inverse of size 5x5
4. determine the inverse of atpa
5. if there is an inverse:
6. pl = prod(m_qweight, m_l)
7. atpl = prod(trans(m_design),pl)
8. m_solution = prod(inverse, atpl)
*)

// pa = prod(m_qweight, m_design)
// [NumDataPts x NumDataPts] . [NumDataPts x Unknowns]
// [NumDataPts x Unknowns]
FOR i := 1 TO GVL.NumberEllipsePoints DO	// rows
	FOR j := 1 TO GVL.Unknowns DO		// columns
		DotProduct := 0;
		FOR k := 1 TO GVL.NumberEllipsePoints DO
			DotProduct := DotProduct + m_qweight[k,i]*m_design[j,k];
		END_FOR
		pa[j,i] := DotProduct;
	END_FOR
END_FOR

// atpa = prod(trans(m_design), pa)
// [Unknown x NumDataPts] . [NumDataPts x Unknown]
// [Unknown x Unknown]
FOR i := 1 TO GVL.Unknowns DO 		// rows
	FOR j := 1 TO GVL.Unknowns DO 	// columns
		DotProduct := 0;
		FOR k := 1 TO GVL.NumberEllipsePoints DO
			DotProduct := DotProduct + m_design[i,k]*pa[j,k];
		END_FOR
		atpa[j,i] := DotProduct;
	END_FOR
END_FOR

// find inverse of atpa
IF Inverse(ADR(atpa),ADR(atpaInverse)) THEN
	// pl = prod(m_qweight, ml) = [NumDataPts x NumDataPts] * [NumDataPts x 1] = [NumDataPts x 1]
	FOR i := 1 TO GVL.NumberEllipsePoints DO			// rows
		DotProduct := 0;
		FOR k := 1 TO GVL.NumberEllipsePoints DO
			DotProduct := DotProduct + m_qweight[k,i]*m_l[k];
		END_FOR
		pl[i] := DotProduct;
	END_FOR
	// atpl = prod(trans(m_design), pl)
	FOR i := 1 TO GVL.Unknowns DO	// rows
		DotProduct := 0;
		FOR k := 1 TO GVL.NumberEllipsePoints DO // columns
			DotProduct := DotProduct + m_design[i,k]*pl[k];
		END_FOR
		atpl[i] := DotProduct;
	END_FOR
	// m_solution = prod(inverse, atpl)
	FOR i := 1 TO GVL.Unknowns DO	// rows
		DotProduct := 0;
		FOR k := 1 TO GVL.Unknowns DO // columns
			DotProduct := DotProduct + atpaInverse[k,i]*atpl[k];
		END_FOR
		m_solutions[i] := DotProduct;
	END_FOR
	EvaluateUnknowns := TRUE;
ELSE
	EvaluateUnknowns := FALSE;
END_IF

_pa := pa;
_atpa := atpa;
_atpaInverse := atpaInverse;
_pl := pl;
_atpl := atpl;
END_METHOD

METHOD FormulateMatrices : BOOL
VAR_INPUT
END_VAR
VAR
	x0		: LREAL;
	y0		: LREAL;
	a		: LREAL;
	b		: LREAL;
	
	sinr	: LREAL;
	cosr	: LREAL;
	asqr	: LREAL;
	bsqr	: LREAL;
	i		: INT;
	x		: LREAL;
	y		: LREAL;
	d1		: LREAL;
	d2		: LREAL;
	p		: LREAL;
	q		: LREAL;
END_VAR
x0 := m_provisionals[1];
y0 := m_provisionals[2];
a := m_provisionals[3];
b := m_provisionals[4];

sinr := SIN(m_provisionals[5]);
cosr := COS(m_provisionals[5]);
asqr := a * a;
bsqr := b * b;

FOR i := 1 TO GVL.NumberEllipsePoints DO
	x := m_observations[1,i];
	y := m_observations[2,i];
	
	d1 := ((y - y0) * cosr - (x - x0)*sinr);
	d2 := ((x - x0) * cosr + (y - y0)*sinr);
	
	m_design[1,i] := 2.0 * ((asqr * d1 * sinr) - (bsqr * d2 * cosr));
	m_design[2,i] := -2.0 * ((bsqr * d2 * sinr) + (asqr * d1 * cosr));
	m_design[3,i] := 2.0 * a * ((d1 * d1) - bsqr);
	m_design[4,i] := 2.0 * b * ((d2 * d2) - asqr);
	m_design[5,i] := 2.0 * d1 * d2 * (bsqr - asqr);
	
	p := 2.0 * ((asqr * d1 * sinr) + (bsqr * d2 * cosr));
	q := -2.0 * ((bsqr * d2 * sinr) + (asqr * d1 * cosr));
	m_qweight[i,i] := 1.0 / (p * p + q * q);
	m_l[i] := -1*((asqr * d1 * d1) + (bsqr * d2 * d2) - (asqr * bsqr));
END_FOR
END_METHOD

METHOD GenerateProvisionals : BOOL
VAR
	_centrex		: LREAL;
	_centrey		: LREAL;
	_dx			: LREAL;
	_dy			: LREAL;
	_major		: LREAL;
	_minor		: LREAL;
	_rotation	: LREAL;
END_VAR
_centrex := 0.5 * (m_maxx + m_minx);
_centrey := 0.5 * (m_maxy + m_miny);
_dx := m_maxx - m_minx;
_dy := m_maxy - m_miny;
IF _dx > _dy THEN
	_major := 0.5 * _dx;
	_minor := 0.5 * _dy;
ELSE
	_major := 0.5 * _dy;
	_minor := 0.5 * _dx;
END_IF
_rotation := ATAN(_dy/_dx);

m_provisionals[1] := _centrex;
m_provisionals[2] := _centrey;
m_provisionals[3] := _major;
m_provisionals[4] := _minor;
m_provisionals[5] := _rotation;
END_METHOD

METHOD HasConverged : BOOL
VAR_INPUT
END_VAR
VAR
	i		: INT;
END_VAR
HasConverged := TRUE;
FOR i := 1 TO GVL.Unknowns DO
	IF ABS(m_solutions[i]) > GVL.ConvergenceCriteria THEN
		HasConverged := FALSE;
	END_IF
END_FOR
END_METHOD

METHOD Inverse : BOOL
VAR_INPUT
	ptrMatrix		: POINTER TO ARRAY[1..5,1..5] OF LREAL;
	ptrInverse		: POINTER TO ARRAY[1..5,1..5] OF LREAL;
END_VAR
VAR
	Determinant		: LREAL;
	Matrix			: ARRAY[1..5,1..5] OF LREAL;
	_Cofactor		: LREAL;
	i				: INT;
	j				: INT;
	SignRow: BOOL;
	SignColumn: BOOL;
END_VAR
IF Determinant5x5(ptrDeterminant := ADR(Determinant), ptrMatrix := ptrMatrix) THEN
	Determinant := 1 / Determinant;
	// get cofactors
	FOR i := 1 TO 5 DO
		FOR j := 1 TO 5 DO
			IF Cofactor(ptrMatrix5x5 := ptrMatrix, ptrCofactor := ADR(_Cofactor), row := i, column := j) THEN
				Matrix[i,j] := _Cofactor;
			ELSE
				Inverse := FALSE;
				RETURN;
			END_IF
		END_FOR
	END_FOR
	_cofactorMatrix := Matrix;
	
	SignRow := TRUE;
	SignColumn := TRUE;
	FOR i := 1 TO 5 DO
		FOR j := 1 TO 5 DO
			IF NOT SignRow THEN
				Matrix[i,j] := (-1) * Matrix[i,j];
			END_IF
			SignRow := NOT SignRow;
		END_FOR
		SignColumn := NOT SignColumn;
		SignRow := SignColumn;
	END_FOR
	_cofactorMatrixSigned := Matrix;
	// transpose 
	Transpose(ADR(Matrix),ptrInverse);
	_cofactorMatrixT := ptrInverse^;
	FOR i := 1 TO 5 DO
		FOR j := 1 TO 5 DO
			ptrInverse^[i,j] := Determinant * ptrInverse^[i,j];
		END_FOR
	END_FOR
	
	Inverse := TRUE;
ELSE
	Inverse := FALSE;
END_IF
END_METHOD

METHOD IsDegenerate : BOOL
VAR_INPUT
	iteration	: INT;
END_VAR
IsDegenerate := (iteration > GVL.MaxIterations);
END_METHOD

PROPERTY major : LREAL
GET
major := m_provisionals[3];

(*
m_provisionals[1] := _centrex;
m_provisionals[2] := _centrey;
m_provisionals[3] := _major;
m_provisionals[4] := _minor;
m_provisionals[5] := _rotation;
*)
END_GET
END_PROPERTY

PROPERTY minor : LREAL
GET
minor := m_provisionals[4];

(*
m_provisionals[1] := _centrex;
m_provisionals[2] := _centrey;
m_provisionals[3] := _major;
m_provisionals[4] := _minor;
m_provisionals[5] := _rotation;
*)
END_GET
END_PROPERTY

METHOD NormalizeAdjustedUnknowns : BOOL
VAR_INPUT
END_VAR
VAR
	theta		: LREAL;
	negative	: BOOL;
	major		: LREAL;
	minor		: LREAL;
END_VAR
theta := ABS(m_provisionals[5]);
negative := m_provisionals[5] < 0;

theta := LMOD(theta, 2*3.14159);
IF negative THEN
	theta := 2*3.14159 - theta;
END_IF

major := m_provisionals[3];
minor := m_provisionals[4];
IF minor > major THEN
	m_provisionals[3] := minor;
	m_provisionals[4] := major;
	theta := theta - (0.5)*3.14159;
	IF theta < 0 THEN
		theta := theta + 2*3.14159;
	END_IF
	m_provisionals[5] := theta;
END_IF
END_METHOD

PROPERTY rotation : LREAL
GET
rotation := m_provisionals[5];

(*
m_provisionals[1] := _centrex;
m_provisionals[2] := _centrey;
m_provisionals[3] := _major;
m_provisionals[4] := _minor;
m_provisionals[5] := _rotation;
*)
END_GET
END_PROPERTY

METHOD Transpose : BOOL
VAR_INPUT
	ptrMatrix		: POINTER TO ARRAY[1..5,1..5] OF LREAL;
	ptrTranspose	: POINTER TO ARRAY[1..5,1..5] OF LREAL;
END_VAR
VAR
	i				: INT;
	j				: INT;
END_VAR
FOR i := 1 TO 5 DO
	FOR j := 1 TO 5 DO
		ptrTranspose^[j,i] := ptrMatrix^[i,j];
	END_FOR
END_FOR
END_METHOD

END_FUNCTION_BLOCK

// ---- POUs/FB_Cutter.TcPOU
FUNCTION_BLOCK FB_Cutter 
VAR_INPUT
END_VAR
VAR_OUTPUT
END_VAR
VAR
	Axis			: AXIS_REF;	// SMAC Actuator
	mcMoveVel		: MC_MoveVelocity;
	mcMoveAbs		: MC_MoveAbsolute;
	mcHome			: MC_Home;
	mcHalt			: MC_Halt;
	mcPower			: MC_Power;
	mcReset			: MC_Reset;
	_errorCode		: UDINT;
	_position		: LREAL;
	_velocity		: LREAL := 20;
	_hmiParameters	: ST_CutterParameters;
	_parameters		: ST_CutterParameters;
	
	fbMessageChange			: FB_TcMessage;
	fbMessageLoaded			: FB_TcMessage;
	
END_VAR

METHOD Abort : BOOL
VAR_INPUT
END_VAR
mcPower(Axis := Axis, Enable := FALSE);
END_METHOD

METHOD Clear : INT
VAR_INPUT
	Execute : BOOL;
END_VAR
VAR_INST
	rTrig	: R_TRIG;
	nIndex	: INT;
END_VAR
rTrig(CLK := Execute);
IF rTrig.Q THEN
	nIndex := 10;
	Reset(Execute := FALSE);
	Home(Execute := FALSE);
	MoveAbs(Execute := FALSE);
END_IF

IF NOT Execute THEN
	nIndex := 0;
END_IF

CASE nIndex OF
	0: // idle state
		Clear := 0;
	10: // reset the cutter
		IF Reset(Execute := TRUE) = 1 THEN
			Reset(Execute := FALSE);
			nIndex := 20;
		END_IF
	20: // enable the cutter
		IF Enable() THEN
			nIndex := 30;
		END_IF
	30: // home the cutter
		IF Home(Execute := TRUE) = 1 THEN
			Home(Execute := FALSE);
			nIndex := 40;
		END_IF
	40: // move to position 5 mm
		_position := 5;
		IF MoveAbs(Execute := TRUE) = 1 THEN
			MoveAbs(Execute := FALSE);
			nIndex := 50;
		END_IF
	50: // done state
		Clear := 1;
END_CASE
END_METHOD

METHOD CutSample : INT
VAR_INPUT
	Execute	: BOOL;
END_VAR
VAR_INST
	rTrig	: R_TRIG;
	nIndex	: INT;
	MoveVelError : BOOL;
	HaltError : BOOL;
	MoveAbsError : BOOL;
	ErrorTimeout	: TON := (PT := T#5s);
END_VAR
rTrig(CLK := Execute);
IF rTrig.Q THEN
	nIndex := 10;
	mcMoveVel(Execute := FALSE, Axis := Axis, BufferMode := MC_BufferMode.MC_Aborting,
		Direction := MC_Direction.MC_Positive_Direction);
	mcMoveAbs(Execute := FALSE, Axis := Axis);
	mcHalt(Execute := FALSE, Axis := Axis);
	mcReset(Execute := FALSE, Axis := Axis);
	ErrorTimeout(IN := FALSE);
	MoveVelError := FALSE;
	HaltError := FALSE;
	MoveAbsError := FALSE;
END_IF

IF NOT Execute THEN
	nIndex := 0;
END_IF

CASE nIndex OF
	0: // idle state
		CutSample := 0;
	10: // make sure its operational
		Axis.ReadStatus();
		IF Axis.Status.Operational THEN
			nIndex := 20;
		END_IF
	20: // make the cut
		mcMoveVel.Execute := TRUE;
		ErrorTimeout.IN := TRUE;
		mcMoveVel.Velocity := _parameters.cutVelocity;
		IF Axis.NcToPlc.ActTorque > 400 THEN
			nIndex := 30;
			mcMoveVel.Execute := FALSE;
			ErrorTimeout.IN := FALSE;
			mcHalt(Axis := Axis, Execute := TRUE);
		END_IF
		IF mcMoveVel.Error THEN
			_errorCode := mcMoveVel.ErrorID;
			ErrorTimeout.IN := FALSE;
			MoveVelError := TRUE;
			nIndex := 70;
		END_IF
		IF ErrorTimeout.Q THEN
			ErrorTimeout.IN := FALSE;
			nIndex := 30;
		END_IF
		ErrorTimeout();
		mcMoveVel(Axis := Axis);
	30: // wait to halt
		mcHalt.Execute := TRUE;
		IF mcHalt.Done THEN
			mcHalt.Execute := FALSE;
			nIndex := 40;
		END_IF
		IF mcHalt.Error THEN
			mcHalt.Execute := FALSE;
			HaltError := TRUE;
			_errorCode := mcHalt.ErrorID;
			nIndex := 70;
		END_IF
		mcHalt(Axis := Axis);
	40: // retract the cutter axis
		mcMoveAbs.Execute := TRUE;
		mcMoveAbs.Position := _parameters.retractPosition;
		mcMoveAbs.Velocity := _parameters.cutVelocity;
		IF mcMoveAbs.Done THEN
			mcMoveAbs.Execute := FALSE;
			nIndex := 50;
		END_IF
		IF mcMoveAbs.Error THEN
			mcMoveAbs.Execute := FALSE;
			MoveAbsError := TRUE;
			_errorCode := mcMoveAbs.ErrorID;
			nIndex := 70;
		END_IF
		mcMoveAbs(Axis := Axis);
	45: // reset the lag
		mcReset.Execute := TRUE;
		IF mcReset.Done THEN
			mcReset.Execute := FALSE;
			nIndex := 50;
		END_IF
		mcReset(Axis := Axis);
	50: // done state
		CutSample := 1;
	70: // error state
		CutSample := -1;
END_CASE
END_METHOD

PROPERTY cutVelocity : LREAL
GET
cutVelocity := _parameters.cutVelocity;
END_GET
SET
fbMessageChange.ipArguments.Clear().AddString('cutVelocity').AddLReal(_parameters.cutVelocity).AddLReal(CutVelocity);
fbMessageChange.Send(0);
_parameters.cutVelocity := cutVelocity;
END_SET
END_PROPERTY

METHOD Disable : BOOL
VAR_INPUT
END_VAR
mcPower(Axis := Axis, Enable := FALSE, Enable_Positive := FALSE, Enable_Negative := FALSE);
Axis.ReadStatus();
Disable := NOT Axis.Status.Operational;
END_METHOD

METHOD Enable : BOOL
VAR_INPUT
END_VAR
mcPower(Axis := Axis, Enable := TRUE, Enable_Positive := TRUE, Enable_Negative := TRUE);
Axis.ReadStatus();
Enable := Axis.Status.Operational;
END_METHOD

METHOD FB_init : BOOL
VAR_INPUT
	bInitRetains : BOOL; // if TRUE, the retain variables are initialized (warm start / cold start)
	bInCopyCode : BOOL;  // if TRUE, the instance afterwards gets moved into the copy code (online change)
END_VAR
IF NOT fbMessageChange.EqualsToEventEntryEx(stOther := TC_EVENTS.SlitterEvents.ParameterChange) THEN
	fbMessageChange.CreateEx(TC_EVENTS.SlitterEvents.ParameterChange, 0);
	fbMessageChange.ipArguments.Clear();
END_IF

IF NOT fbMessageLoaded.EqualsToEventEntryEx(stOther := TC_EVENTS.SlitterEvents.ParametersLoadedFromFile) THEN
	fbMessageLoaded.CreateEx(TC_EVENTS.SlitterEvents.ParametersLoadedFromFile, 0);
	fbMessageLoaded.ipArguments.Clear().AddString('Cutter');
END_IF
END_METHOD

METHOD Home : INT
VAR_INPUT
	Execute	: BOOL;
END_VAR
VAR_INST
	rTrig	: R_TRIG;
	nIndex	: INT;
	PosDif	: LREAL;
END_VAR
rTrig(CLK := Execute);
IF rTrig.Q THEN
	nIndex := 10;
	mcMoveVel(Axis := Axis, Execute := FALSE, Direction := MC_Direction.MC_Negative_Direction);
	mcHalt(Axis := Axis, Execute := FALSE);
	mcHome(Axis := Axis, Execute := FALSE);
END_IF

IF NOT Execute THEN
	nIndex := 0;
END_IF

CASE nIndex OF
	0: // idle state
		Home := 0;
	10: // move up (negative direction) slowly, watch the pos dif
		mcMoveVel.Execute := TRUE;
		IF mcMoveVel.InVelocity THEN
			mcMoveVel.Execute := FALSE;
			nIndex := 15;
		END_IF
		IF mcMoveVel.Error THEN
			mcMoveVel.Execute := FALSE;
			_errorCode := mcMoveVel.ErrorID;
			nIndex := 50;
		END_IF
	15: // 
		IF Axis.NcToPlc.PosDiff < -1 THEN
			PosDif := Axis.NcToPlc.PosDiff;
			mcHalt.Execute := TRUE;
			nIndex := 20;
		END_IF
		IF mcMoveVel.Error THEN
			mcMoveVel.Execute := FALSE;
			_errorCode := mcMoveVel.ErrorID;
			nIndex := 50;
		END_IF
	20: // wait for halt to finish
		IF mcHalt.Done THEN
			mcHalt.Execute := FALSE;
			nIndex := 30;
		END_IF
		IF mcHalt.Error THEN
			mcHalt.Execute := FALSE;
			_errorCode := mcHalt.ErrorID;
			nIndex := 50;
		END_IF
	30: // set this position as -1
		mcHome.Execute := TRUE;
		mcHome.HomingMode := MC_Direct;
		mcHome.Position := -1;
		IF mcHome.Done THEN
			mcHome.Execute := FALSE;
			nIndex := 40;
		END_IF
		IF mcHome.Error THEN
			mcHome.Execute := FALSE;
			_errorCode := mcHome.ErrorID;
			nIndex := 50;
		END_IF
	40: // done
		Home := 1;
	50: // error state 
		Home := -1;		

END_CASE

mcMoveVel(
	Axis := Axis, 
	Velocity := 5, 
	Direction := MC_Direction.MC_Negative_Direction);
mcHalt(Axis := Axis);
mcHome(Axis := Axis);
END_METHOD

PROPERTY IsEnabled : BOOL
GET
Axis.ReadStatus();
IsEnabled := Axis.Status.Operational;
END_GET
END_PROPERTY

METHOD MonitorParameters : BOOL
VAR_INPUT
END_VAR
IF _hmiParameters.cutVelocity <> cutVelocity THEN
	cutVelocity := _hmiParameters.cutVelocity;
END_IF

IF _hmiParameters.retractPosition <> retractPosition THEN
	retractPosition := _hmiParameters.retractPosition;
END_IF
END_METHOD

METHOD MoveAbs : INT
VAR_INPUT
	Execute	: BOOL;
END_VAR
VAR_INST
	nIndex 	: INT;
	rTrig	: R_TRIG;
END_VAR
rTrig(CLK := Execute);
IF rTrig.Q THEN
	nIndex := 10;
	mcMoveAbs(Axis := Axis, Execute := FALSE);
END_IF

IF NOT Execute THEN
	nIndex := 0;
END_IF

CASE nIndex OF
	0: // idle state
		MoveAbs := 0;
	10: // move
		mcMoveAbs.Execute := TRUE;
		mcMoveAbs.Position := _position;
		mcMoveAbs.Velocity := _velocity;
		IF mcMoveAbs.Done THEN
			nIndex := 20;
			mcMoveAbs.Execute := FALSE;
		END_IF
		IF mcMoveAbs.Error THEN
			nIndex := 30;
			_errorCode := mcMoveAbs.ErrorID;
			mcMoveAbs.Execute := FALSE;
		END_IF
		mcMoveAbs(Axis := Axis);
	20: // done state
		MoveAbs := 1;
	30: // error state
		MoveAbs := -1;
END_CASE
END_METHOD

PROPERTY Parameters : ST_CutterParameters
GET
Parameters := _parameters;
END_GET
SET
fbMessageLoaded.Send(0);
_parameters := Parameters;
_hmiParameters := Parameters;
END_SET
END_PROPERTY

METHOD Reset : INT
VAR_INPUT
	Execute	: BOOL;
END_VAR
VAR_INST
	nIndex 	: INT;
	rTrig	: R_TRIG;
END_VAR
rTrig(CLK := Execute);
IF rTrig.Q THEN
	nIndex := 10;
	mcReset(Axis := Axis, Execute := FALSE);
	Home(Execute := FALSE);
	mcMoveAbs(Axis := Axis, Execute := FALSE);
	mcHome(Axis := Axis, Execute := FALSE);
	mcMoveVel(Axis := Axis, Execute := FALSE);
	mcHalt(Axis := Axis, Execute := FALSE);		
	_errorCode := 0;
END_IF

IF NOT Execute THEN
	nIndex := 0;
END_IF

Axis.ReadStatus();

CASE nIndex OF
	0: // idle state
		Reset := 0;
	10: // reset the motor
		IF Disable() THEN
			nIndex := 20;
		END_IF
	20: // check if there is an error
		IF Axis.Status.Error THEN
			nIndex := 30;
		ELSE
			nIndex := 40;
		END_IF
	30: // reset the axis
		mcReset.Execute := TRUE;
		IF mcReset.Done THEN
			nIndex := 40;
			mcReset.Execute := FALSE;
		END_IF
		mcReset(Axis := Axis);
	40: // enable the drive
		IF Enable() THEN
			nIndex := 60;
		END_IF
	60: // done state
		Reset := 1;
	70: // error state
		Reset := -1;
END_CASE
END_METHOD

PROPERTY retractPosition : LREAL
GET
retractPosition := _parameters.retractPosition;
END_GET
SET
fbMessageChange.ipArguments.Clear().AddString('retractPosition').AddLReal(_parameters.retractPosition).AddLReal(retractPosition);
fbMessageChange.Send(0);
_parameters.retractPosition := retractPosition;
END_SET
END_PROPERTY

END_FUNCTION_BLOCK

// ---- POUs/FB_Ejector.TcPOU
FUNCTION_BLOCK FB_Ejector
VAR_INPUT
END_VAR
VAR_OUTPUT
END_VAR
VAR	
	axis					: FB_Axis;
	zSlide					: FB_Actuator;	
	_Vacuum AT %Q*			: BOOL;
	_VacuumSensor AT %I*	: BOOL;
	_BlowOff AT %Q*			: BOOL;
	_hmiParameters			: ST_EjectorParameters;
	_parameters				: ST_EjectorParameters;
	
	fbMessageChange			: FB_TcMessage;
	fbMessageLoaded			: FB_TcMessage;
	
END_VAR

METHOD Abort : BOOL
VAR_INPUT
END_VAR
BlowOff := FALSE;
PickUpVacuum := FALSE;
zSlide.Neutral();
axis.Disable();
EjectSamplePass(Execute := FALSE);
EjectSampleFail(Execute := FALSE);
Reset(Execute := FALSE);
END_METHOD

PROPERTY BlowOff : BOOL
GET
BlowOff := _BlowOff;
END_GET
SET
_BlowOff := BlowOff;
END_SET
END_PROPERTY

PROPERTY EjectAxisFailPosition : LREAL
GET
EjectAxisFailPosition := _parameters.ejectPositionFail;
END_GET
SET
fbMessageChange.ipArguments.Clear().AddString('EjectAxisFailPosition').AddLReal(_parameters.ejectPositionFail).AddLReal(EjectAxisFailPosition);
fbMessageChange.Send(0);
_parameters.ejectPositionFail := EjectAxisFailPosition;
END_SET
END_PROPERTY

PROPERTY EjectAxisHomePosition : LREAL
GET
EjectAxisHomePosition := _parameters.ejectPositionHome;
END_GET
SET
fbMessageChange.ipArguments.Clear().AddString('EjectAxisHomePosition').AddLReal(_parameters.ejectPositionHome).AddLReal(EjectAxisHomePosition);
fbMessageChange.Send(0);
_parameters.ejectPositionHome := EjectAxisHomePosition;
END_SET
END_PROPERTY

PROPERTY EjectAxisPassPosition : LREAL
GET
EjectAxisPassPosition := _parameters.ejectPositionPass;
END_GET
SET
fbMessageChange.ipArguments.Clear().AddString('EjectAxisPassPosition').AddLReal(_parameters.ejectPositionPass).AddLReal(EjectAxisPassPosition);
fbMessageChange.Send(0);
_parameters.ejectPositionPass := EjectAxisPassPosition;
END_SET
END_PROPERTY

PROPERTY EjectAxisVelocity : LREAL
GET
EjectAxisVelocity := _parameters.ejectVelocity;
END_GET
SET
fbMessageChange.ipArguments.Clear().AddString('EjectAxisVelocity').AddLReal(_parameters.ejectVelocity).AddLReal(EjectAxisVelocity);
fbMessageChange.Send(0);
_parameters.ejectVelocity := EjectAxisVelocity;
END_SET
END_PROPERTY

METHOD EjectSampleFail : INT
VAR_INPUT
	Execute	: BOOL;
END_VAR
VAR_INST
	rTrig	: R_TRIG;
	nIndex	: INT;
	TON		: TON;
	Message	: STRING(255);
END_VAR
VAR
	
END_VAR
EjectSampleFail := 0;
rTrig(CLK := Execute);
IF rTrig.Q THEN
	axis.AbsMove(Execute := FALSE, Position := 0, Velocity := 0);
	nIndex := 10;
END_IF

IF NOT Execute THEN
	nIndex := 0;
END_IF

CASE nIndex OF
	10: // verify that we are retracted in x
		Message := 'Moving to pick up location';
		IF axis.AbsMove(Execute := TRUE, Position := _parameters.ejectPositionHome, Velocity := _parameters.ejectVelocity) THEN
			axis.AbsMove(Execute := FALSE, Position := 0, Velocity := 0);
			nIndex := 20;
		END_IF
		IF axis.Error THEN
			Message := 'Error moving to pick up location';
			axis.AbsMove(Execute := FALSE, Position := 0, Velocity := 0);
			nIndex := 911;
		END_IF
	20: // extend z axis turn on pick up vacuum
		Message := 'Extending z actuator';
		_Vacuum := TRUE;
		IF zSlide.Extend() = 1 THEN
			nIndex := 30;	
		ELSIF zSlide.Extend() = -1 THEN
			Message := 'Error extending z actuator';
			nIndex := 911;
		END_IF
	30: // wait a second
		TON.IN := TRUE;
		TON.PT := T#750MS;
		IF TON.Q THEN
			TON.IN := FALSE;
			nIndex := 40;
		END_IF
		TON();
	40: // retract z axis
		Message := 'Retract z actuator';
		IF zSlide.Retract() = 1 THEN
			nIndex := 50;
		ELSIF zSlide.Retract() = -1 THEN
			Message := 'Error retracting z actuaor';
			nIndex := 911;
		END_IF
	50: // extend the x axis; turn on the blowoff air
		Message := 'Moving to eject reject position';
		IF axis.AbsMove(Execute := TRUE, Position := _parameters.ejectPositionFail, Velocity := _parameters.ejectVelocity) THEN
			axis.AbsMove(Execute := FALSE, Position := 0, Velocity := 0);
			nIndex := 60;
		END_IF
		IF axis.Error THEN
			Message := 'Error moving to reject position';
			nIndex := 911;
			axis.AbsMove(Execute := FALSE, Position := 0, Velocity := 0);
		END_IF
	60: // turn off the blow off	
		_Vacuum := FALSE;	
		IF zSlide.Extend() = 1 THEN
			_BlowOff := TRUE;
		END_IF
		TON.IN := _BlowOff;
		TON.PT := T#500MS;
		IF TON.Q THEN
			_BlowOff := FALSE;		
			TON.IN := FALSE;
			nIndex := 70;
		END_IF
		TON();
	70: // retract the x axis
		Message := 'Moving back to pick up position.';
		zSlide.Retract();
		IF axis.AbsMove(Execute := TRUE, Position := _parameters.ejectPositionHome, Velocity := _parameters.ejectVelocity) THEN
			axis.AbsMove(Execute := FALSE, Position := 0, Velocity := 0);
			nIndex := 80;
		END_IF
		IF axis.Error THEN
			Message := 'Error moving back to pick up position';
			axis.AbsMove(Execute := FALSE, Position := 0, Velocity := 0);
			nIndex := 911;
		END_IF
	80: // done state
		EjectSampleFail := 1;		
END_CASE
END_METHOD

METHOD EjectSamplePass : INT
VAR_INPUT
	Execute	: BOOL;
END_VAR
VAR_INST
	rTrig	: R_TRIG;
	nIndex	: INT;
	TON		: TON;
	Message	: STRING;
END_VAR
EjectSamplePass := 0;
rTrig(CLK := Execute);
IF rTrig.Q THEN
	axis.AbsMove(Execute := FALSE, Position := 0, Velocity := 0);
	nIndex := 10;
END_IF

IF NOT Execute THEN
	nIndex := 0;
END_IF

CASE nIndex OF
	10: // verify that we are retracted in x
		Message := 'Moving to pick up location';
		IF axis.AbsMove(Execute := TRUE, Position := _parameters.ejectPositionHome, Velocity := _parameters.ejectVelocity) THEN
			axis.AbsMove(Execute := FALSE, Position := 0, Velocity := 0);
			nIndex := 20;
		END_IF
		IF axis.Error THEN
			Message := 'Error moving to pick up location';
			axis.AbsMove(Execute := FALSE, Position := 0, Velocity := 0);
			nIndex := 911;
		END_IF
	20: // extend z axis turn on pick up vacuum
		Message := 'Extending z actuator';
		_Vacuum := TRUE;
		IF zSlide.Extend() = 1 THEN
			nIndex := 30;
		ELSIF zSlide.Extend() = -1 THEN
			Message := 'Error extending z actuator';
			nIndex := 911;
		END_IF
	30: // wait a second
		TON.IN := TRUE;
		TON.PT := T#750MS;
		IF TON.Q THEN
			TON.IN := FALSE;
			nIndex := 40;
		END_IF
		TON();
	40: // retract z axis
		Message := 'Retract z actuator';
		IF zSlide.Retract() = 1 THEN
			nIndex := 50;
		ELSIF zSlide.Retract() = -1 THEN
			Message := 'Error retracting z actuaor';
			nIndex := 911;
		END_IF		
	50: // extend the x axis; turn on the blowoff air
		Message := 'Moving to eject pass position';
		IF axis.AbsMove(Execute := TRUE, Position := _parameters.ejectPositionPass, Velocity := _parameters.ejectVelocity) THEN
			axis.AbsMove(Execute := FALSE, Position := 0, Velocity := 0);
			nIndex := 60;
		END_IF
		IF axis.Error THEN
			Message := 'Error moving to pass position';
			nIndex := 911;
			axis.AbsMove(Execute := FALSE, Position := 0, Velocity := 0);
		END_IF
	60: // turn off the blow off		
		_Vacuum := FALSE;
		IF zSlide.Extend() = 1 THEN
			_BlowOff := TRUE;	
		END_IF
		TON.IN := _BlowOff;
		TON.PT := T#500MS;
		IF TON.Q THEN
			_BlowOff := FALSE;		
			TON.IN := FALSE;
			nIndex := 70;
		END_IF
		TON();
	70: // retract the x axis
		Message := 'Moving back to pick up position.';
		zSlide.Retract();
		IF axis.AbsMove(Execute := TRUE, Position := _parameters.ejectPositionHome, Velocity := _parameters.ejectVelocity) THEN
			axis.AbsMove(Execute := FALSE, Position := 0, Velocity := 0);
			nIndex := 80;
		END_IF
		IF axis.Error THEN
			Message := 'Error moving back to pick up position';
			axis.AbsMove(Execute := FALSE, Position := 0, Velocity := 0);
			nIndex := 911;
		END_IF
	80: // done state
		EjectSamplePass := 1;		
END_CASE
END_METHOD

METHOD FB_init : BOOL
VAR_INPUT
	bInitRetains : BOOL; // if TRUE, the retain variables are initialized (warm start / cold start)
	bInCopyCode : BOOL;  // if TRUE, the instance afterwards gets moved into the copy code (online change)
END_VAR
IF NOT fbMessageChange.EqualsToEventEntryEx(stOther := TC_EVENTS.SlitterEvents.ParameterChange) THEN
	fbMessageChange.CreateEx(TC_EVENTS.SlitterEvents.ParameterChange, 0);
	fbMessageChange.ipArguments.Clear();
END_IF

IF NOT fbMessageLoaded.EqualsToEventEntryEx(stOther := TC_EVENTS.SlitterEvents.ParametersLoadedFromFile) THEN
	fbMessageLoaded.CreateEx(TC_EVENTS.SlitterEvents.ParametersLoadedFromFile, 0);
	fbMessageLoaded.ipArguments.Clear().AddString('Ejector');
END_IF
END_METHOD

PROPERTY IsEjectZExtend : BOOL
GET
IsEjectZExtend := zSlide.IsExtended;
END_GET
END_PROPERTY

PROPERTY IsEjectZRetract : BOOL
GET
IsEjectZRetract := zSlide.IsRetracted;
END_GET
END_PROPERTY

METHOD MonitorParameters : BOOL
VAR_INPUT
END_VAR
IF _hmiParameters.ejectPositionFail <> EjectAxisFailPosition THEN
	EjectAxisFailPosition := _hmiParameters.ejectPositionFail;
END_IF

IF _hmiParameters.ejectPositionHome <> EjectAxisHomePosition THEN
	EjectAxisHomePosition := _hmiParameters.ejectPositionHome;
END_IF

IF _hmiParameters.ejectPositionPass <> EjectAxisPassPosition THEN
	EjectAxisPassPosition := _hmiParameters.ejectPositionPass;
END_IF

IF _hmiParameters.ejectVelocity <> EjectAxisVelocity THEN
	EjectAxisVelocity := _hmiParameters.ejectVelocity;
END_IF
END_METHOD

PROPERTY Parameters : ST_EjectorParameters
GET
Parameters := _parameters;
END_GET
SET
fbMessageLoaded.Send(0);
_parameters := Parameters;
_hmiParameters := Parameters;
END_SET
END_PROPERTY

PROPERTY PickUpVacuum : BOOL
GET
PickUpVacuum := _Vacuum;
END_GET
SET
_Vacuum := PickUpVacuum;
END_SET
END_PROPERTY

METHOD Reset : INT
VAR_INPUT
	Execute	: BOOL;
END_VAR
VAR_INST
	rTrig	: R_TRIG;
	nIndex	: INT;
END_VAR
Reset := 0;

rTrig(CLK := Execute);
IF rTrig.Q THEN
	nIndex := 5;
	EjectSampleFail(Execute := FALSE);
	EjectSamplePass(Execute := FALSE);
	axis.AbsMove(Execute := FALSE, Position := 0, Velocity := 0);
	axis.Reset(Execute := FALSE);
END_IF

IF NOT Execute THEN
	nIndex := 0;
END_IF

CASE nIndex OF
	5: 
		BlowOff := FALSE;
		PickUpVacuum := FALSE;
		zSlide.Reset();
		nIndex := 7;
	7: // retract the z axis
		IF zSlide.Retract() = 1 THEN
			nIndex := 10;
		ELSIF zSlide.Retract() = -1 THEN
			nIndex := 911;
		END_IF
		
	10: // disable the axis
		IF axis.Disable() THEN
			nIndex := 20;
		END_IF
	20: // check if there's an error
		IF axis.Error THEN
			nIndex := 30;
		ELSE
			nIndex := 40;
		END_IF
	30: // reset the drive
		IF axis.Reset(Execute := TRUE) THEN
			axis.Reset(Execute := FALSE);
			nIndex := 20;
		END_IF
	40: // enable the drive
		IF axis.Enable() THEN
			nIndex := 50;
		END_IF
	50: // move to the home position
		IF axis.AbsMove(Execute := TRUE, Position := _parameters.ejectPositionHome, Velocity := _parameters.ejectVelocity) THEN
			axis.AbsMove(Execute := FALSE, Position := 0, Velocity := 0);
			nIndex := 60;
		END_IF
		IF axis.Error THEN
			axis.AbsMove(Execute := TRUE, Position := 0, Velocity := 0);
			nIndex := 911;
		END_IF
	60: // done state
		Reset := 1;		
END_CASE
END_METHOD

METHOD ReturnToIdle : INT
VAR_INPUT
END_VAR
_BlowOff := FALSE;
_Vacuum := FALSE;
END_METHOD

END_FUNCTION_BLOCK

// ---- POUs/FB_Actuator.TcPOU
FUNCTION_BLOCK FB_Actuator IMPLEMENTS I_Actuator
VAR_INPUT
END_VAR
VAR_OUTPUT
END_VAR
VAR
	doValveExtend AT %Q*	: BOOL;
	doValveRetract AT %Q*	: BOOL;
	diRetracted AT %I*		: BOOL;
	diExtended AT %I*		: BOOL;
	ExtendTon				: TON := (PT := T#5S);
	RetractTon				: TON := (PT := T#5S);
	fbExtendAlarm			: FB_TcAlarm;
	fbRetractAlarm			: FB_TcAlarm;
END_VAR

PROPERTY Error : BOOL
GET
END_GET
SET
END_SET
END_PROPERTY

METHOD Extend : INT
VAR_INPUT
END_VAR
Extend := 0;
doValveExtend := TRUE;
doValveRetract := FALSE;
ExtendTon(IN := NOT diExtended);
IF diExtended THEN
	ExtendTon(IN := FALSE);
	IF fbExtendAlarm.bRaised THEN
		fbExtendAlarm.Clear(0, FALSE);
	END_IF
	Extend := 1;
END_IF
IF ExtendTon.Q THEN
	ExtendTON(IN := FALSE);
	fbExtendAlarm.Raise(0);
	Extend := -1;
END_IF
END_METHOD

METHOD FB_init : BOOL
VAR_INPUT
	bInitRetains : BOOL; // if TRUE, the retain variables are initialized (warm start / cold start)
	bInCopyCode : BOOL;  // if TRUE, the instance afterwards gets moved into the copy code (online change)
END_VAR
IF NOT fbExtendAlarm.EqualsToEventEntryEx(stOther := TC_EVENTS.SlitterEvents.ZActuatorExtendError) THEN
	fbExtendAlarm.CreateEx(TC_EVENTS.SlitterEvents.ZActuatorExtendError, FALSE, 0);
END_IF
IF NOT fbRetractAlarm.EqualsToEventEntryEx(stOther := TC_EVENTS.SlitterEvents.ZActuatorRetractError) THEN
	fbRetractAlarm.CreateEx(TC_EVENTS.SlitterEvents.ZActuatorRetractError, FALSE, 0);
END_IF
END_METHOD

PROPERTY IsExtended : BOOL
GET
IsExtended := diExtended;
END_GET
END_PROPERTY

PROPERTY IsRetracted : BOOL
GET
IsRetracted := diRetracted;
END_GET
END_PROPERTY

METHOD Neutral : BOOL
VAR_INPUT
END_VAR
doValveExtend := FALSE;
doValveRetract := FALSE;
Neutral := TRUE;
END_METHOD

METHOD Reset : BOOL
VAR_INPUT
END_VAR
IF fbExtendAlarm.bRaised THEN
	fbExtendAlarm.Clear(0, FALSE);
END_IF
IF fbRetractAlarm.bRaised THEN
	fbRetractAlarm.Clear(0, FALSE);
END_IF
ExtendTon(IN := FALSE);
RetractTon(IN := FALSE);
END_METHOD

METHOD Retract : INT
VAR_INPUT
END_VAR
Retract := 0;
doValveExtend := FALSE;
doValveRetract := TRUE;
RetractTon(IN := NOT diRetracted);
IF diRetracted THEN
	RetractTon(IN := FALSE);
	IF fbRetractAlarm.bRaised THEN
		fbRetractAlarm.Clear(0, FALSE);
	END_IF
	Retract := 1;
END_IF
IF RetractTon.Q THEN
	RetractTon(IN := FALSE);
	fbRetractAlarm.Raise(0);
	Retract := -1;
END_IF
END_METHOD

END_FUNCTION_BLOCK

// ---- POUs/FB_Frame.TcPOU
FUNCTION_BLOCK FB_Frame IMPLEMENTS I_Frame
VAR_INPUT
END_VAR
VAR_OUTPUT
END_VAR
VAR
	diControlLeft	AT %I*	: BOOL;		// start button left
	diControlRight	AT %I*	: BOOL;		// start button right
	doGreen			AT %Q*	: BOOL;		// solid = ready to start; blinking = sample missing on vacuum
	diDoor1			AT %I*	: BOOL;		// door closed indicator
	diDoor2 		AT %I*	: BOOL;		// door closed indicator
	diDoor3			AT %I*	: BOOL;		// door closed indicator
	diDoor4			AT %I*	: BOOL;		// door closed indicator
	aiPressure		AT %I*	: INT;		// pressure to the system	
	GreenTon				: TON := (PT := T#1S);
	_pressure				: LREAL;
END_VAR

METHOD BlinkGreen : BOOL
VAR_INPUT
END_VAR
VAR_INST
	TonGreen	: TON := (PT := T#1s);
END_VAR
TONGreen.IN := NOT TONGreen.Q;
TONGreen();
IF TONGreen.Q THEN
	GreenLight := NOT GreenLight;
END_IF
END_METHOD

PROPERTY ControlLeft : BOOL
GET
ControlLeft := diControlLeft;
END_GET
END_PROPERTY

PROPERTY ControlRight : BOOL
GET
ControlRight := diControlRight;
END_GET
END_PROPERTY

PROPERTY Door1 : BOOL
GET
Door1 := diDoor1;
END_GET
END_PROPERTY

PROPERTY Door2 : BOOL
GET
Door2 := diDoor2;
END_GET
END_PROPERTY

PROPERTY Door3 : BOOL
GET
Door3 := diDoor3;
END_GET
END_PROPERTY

PROPERTY Door4 : BOOL
GET
Door4 := diDoor4;
END_GET
END_PROPERTY

PROPERTY GreenLight : BOOL
GET
GreenLight := doGreen;
END_GET
SET
doGreen := GreenLight;
END_SET
END_PROPERTY

PROPERTY Pressure : LREAL
GET
VAR
	Slope	: LREAL;
	Intercept : LREAL;
END_VAR
// 1 V = 0PSIG
// 5V = 145 PSIG
Slope := 145 / 4;
Intercept := 145 / 4.0;
Pressure := Slope * (INT_TO_LREAL(aiPressure) * 10 / 32767) - Intercept;
_pressure := Pressure;
END_GET
END_PROPERTY

END_FUNCTION_BLOCK

// ---- Ellipse/FB_ComputeFromImage.TcPOU
FUNCTION_BLOCK FB_ComputeFromImage
VAR_INPUT
	ptrXValues	: POINTER TO ARRAY[1..GVL.NumberVisionPoints] OF REAL;
	ptrYValues	: POINTER TO ARRAY[1..GVL.NumberVisionPoints] OF REAL;
	minor		: LREAL;	// in mm
	pitch		: LREAL;	// mm per pixel
END_VAR
VAR_OUTPUT
	centerX		: LREAL;
	centerY		: LREAL;
	a			: LREAL;	// major in mm
	b			: LREAL;	// minor in mm
END_VAR
	
VAR
	fbSecond	: FB_SecondOrder;
	fbFourth	: FB_FourthOrder;
	fbEllipse	: FB_Ellipse;
	xPeak		: LREAL;
	yPeak		: LREAL;
	XMirror		: ARRAY[1..GVL.NumberEllipsePoints] OF LREAL;
	YMirror		: ARRAY[1..GVL.NumberEllipsePoints] OF LREAL;
	CenterLine	: LREAL;
	i			: INT;
END_VAR

fbSecond.FindPeak(xValues := ptrXValues, yValues := ptrYValues, xPeak := ADR(xPeak));
fbFourth.FindYatX(xValues := ptrXValues, yValues := ptrYValues, xPeak := ADR(xPeak), yPeak := ADR(yPeak));
centerLine := yPeak - (minor / pitch);

FOR i := 1 TO GVL.NumberVisionPoints DO
	XMirror[i] := REAL_TO_LREAL(ptrXValues^[i]);	
	XMirror[i + GVL.NumberVisionPoints] := REAL_TO_LREAL(ptrXValues^[i]);
	YMirror[i] := REAL_TO_LREAL(ptrYValues^[i]);
	YMirror[i + GVL.NumberVisionPoints] := REAL_TO_LREAL(ptrYValues^[i] - ABS(2*(ptrYValues^[i] - centerLine)));
END_FOR

fbEllipse.EllipseFit(xValues := xMirror, yValues := yMirror);
centerX := fbEllipse.centrex;
centerY := fbEllipse.centrey;
a := fbEllipse.major * pitch;
b := fbEllipse.minor * pitch;

END_FUNCTION_BLOCK

// ---- GlobalTextList.TcGTLO
TEXTLIST GlobalTextList
  172 = '\tTube Cutting and Inspection System'
  301 = '    Tube Cutting and Inspection System'
  353 = '    Tube Cutting and Inspection System       '
  1384 = '%0.1f'
  965 = '%0.2f'
  1097 = '%0.2f deg'
  358 = '%0.2f mmHg'
  162 = '%0.3f mm'
  205 = '%d'
  2490 = '%s'
  362 = 'ABORT'
  725 = 'ActPos = %0.2f mm'
  312 = 'ActVel = %0.2f mm/s'
  1624 = 'Air System'
  951 = 'angle = %0.2f deg'
  1389 = 'Assembly Commands'
  963 = 'Axis Error = %d'
  2298 = 'Batch '
  900 = 'Blob Center (col) = %0.2f px'
  1783 = 'Blob Center (row) = %0.2f px'
  1763 = 'Blob delta(column) = %0.2f px'
  553 = 'Blob delta(row) = %0.2f px'
  1787 = 'Blob Height = %0.2f px'
  751 = 'Blob Length = %0.2f px'
  259 = 'Calibrate Camera'
  947 = 'Calibrate Cut Position'
  1470 = 'Calibrate Mandrel'
  287 = 'Calibration Parameters and Results'
  136 = 'Camera'
  2485 = 'Camera Angle'
  190 = 'Camera Control'
  1086 = 'Change Password'
  1297 = 'Column = %0.2f px'
  851 = 'Commands'
  336 = 'Compute'
  1620 = 'Count = %0.0f'
  967 = 'Current Position = %0.2f deg'
  398 = 'Current Position = %0.2f mm'
  1843 = 'Current Position = %0.2f mm/s'
  2143 = 'Cut Distance from Center (mm) for X and Y'
  11 = 'Cut Height'
  666 = 'Cut Length'
  260 = 'Cut Position'
  2291 = 'Cut Position Tolerance'
  647 = 'Cut Results'
  482 = 'Cut Sample'
  914 = 'Cut Velocity = %0.2f mm/s'
  803 = 'Cutter'
  2144 = 'cutter = %0.2f mm'
  174 = 'cutter = %0.2f mm/s'
  1056 = 'Cutter Angle'
  625 = 'Cutter Control'
  1255 = 'Cutter Retract'
  1395 = 'Decrement Spindle'
  848 = 'Description'
  964 = 'Detection Adjustment'
  1927 = 'Diameter'
  937 = 'distance = %0.2f mm'
  2843 = 'Door 1'
  1997 = 'Door 2'
  280 = 'Door 3'
  1431 = 'Door 4'
  785 = 'Edge Detection'
  530 = 'Edit Users'
  616 = 'Eject Position'
  92 = 'Eject Positions'
  347 = 'Eject Sample'
  651 = 'Eject Sample Fail'
  1311 = 'Eject Sample Pass'
  313 = 'Ejector'
  1875 = 'ejector = %0.2f mm/s'
  688 = 'Ejector Commands'
  525 = 'Ejector Control'
  1941 = 'Ejector Reset'
  978 = 'Enable/Disable '
  968 = 'Enable/Disable Axis'
  1502 = 'Enable/Disable X'
  506 = 'Error'
  860 = 'Error Spindle = %d'
  469 = 'Error X = %d'
  217 = 'Error Y = %d'
  749 = 'Exit'
  137 = 'Extend X Axis'
  983 = 'Extend Z Axis'
  1523 = 'Failed'
  2687 = 'FAILED'
  1148 = 'for'
  408 = 'Frame'
  131 = 'Frame '
  894 = 'Height = %0.2f px'
  520 = 'Home'
  794 = 'Inc = %0.2f degrees'
  988 = 'Increment Spindle'
  2749 = 'Initializing'
  1537 = 'Inspect'
  957 = 'Inspect Position'
  80 = 'Inspect Sample'
  37 = 'Inspection Criteria'
  211 = 'Inspection Results'
  2484 = 'Inspection without Compensation '
  2596 = 'Left Finger Switch'
  104 = 'length = %0.2f mm'
  1018 = 'Length = %0.3f mm'
  316 = 'Load Position'
  1065 = 'Load Positions'
  706 = 'Location'
  1363 = 'Login'
  839 = 'Lower the Mandrel'
  2848 = 'Machine Parameters'
  1538 = 'Machine Settings'
  2455 = 'Machine Status'
  258 = 'Mandrel'
  379 = 'Mandrel Control'
  201 = 'Mandrel Vacuum'
  708 = 'Manual '
  2224 = 'Manual Control'
  33 = 'Manual Inspection'
  1169 = 'Max = %0.2f mm'
  82 = 'Min = %0.2f mm'
  314 = 'mm per px (col) = %0.4f'
  1885 = 'mm per px (row) = %0.4f'
  476 = 'Motion Error = %d'
  795 = 'Move Absolute'
  299 = 'Move Axis'
  328 = 'Move To Cut Position'
  88 = 'Move To Eject Position'
  389 = 'Move To Inspect Position'
  100 = 'Move To Load Position'
  415 = 'Move To Pass'
  1118 = 'Move To Pick Up'
  1894 = 'Move To Reject'
  742 = 'Move Vacuum Axis'
  39 = 'Neutral X Axis'
  663 = 'Neutral Z Axis '
  583 = 'No Image Detected'
  552 = 'Operation'
  872 = 'Part Count'
  2012 = 'Part Diameter = %0.2f mm'
  556 = 'Part Pocket Depth = %0.2f mm'
  399 = 'pass = %0.2f mm'
  1639 = 'Pass Position = %0.2f mm'
  1945 = 'Pass Position = %0.2f mm/s'
  1627 = 'PASSED'
  1216 = 'Pattern Match'
  852 = 'Peak (col) = %0.2f px'
  1402 = 'Peak (row) = %0.2f px'
  111 = 'pick up = %0.2f mm'
  853 = 'Pick Up Position = %0.2f mm'
  1237 = 'Pick Up Position = %0.2f mm/s'
  1584 = 'Pocket Depth'
  637 = 'Position = %0.2f mm'
  1324 = 'Pressure (PSIG):'
  1133 = 'Processing'
  1762 = 'Product Code'
  1284 = 'Product Dimensions'
  2416 = 'Product Selection'
  2364 = 'Product Settings'
  896 = 'Raise the Mandrel'
  101 = 'Raw Data'
  2390 = 'Ready'
  401 = 'reject = %0.2f mm'
  2075 = 'Reject Position = %0.2f mm'
  1351 = 'Reject Position = %0.2f mm/s'
  822 = 'Reset'
  1561 = 'RESET'
  1383 = 'Reset Axis'
  241 = 'Reset Motors'
  1964 = 'Reset Vacuum Axis'
  81 = 'Retract Position = %0.2f mm'
  19 = 'Retract X Axis'
  248 = 'Retract Z Axis'
  180 = 'Return Tube'
  502 = 'Right Finger Switch'
  1149 = 'Row = %0.2f px'
  1218 = 'Running'
  1943 = 'Save'
  1105 = 'Save Parameters'
  338 = 'Selection'
  537 = 'spindle = %0.2f mm/s'
  498 = 'Spindle Enable Toggle'
  1285 = 'Spindle Increment (degrees):'
  551 = 'Status = %s'
  703 = 'Subassembly'
  213 = 'Target Torque = %d %% MaxTorque'
  194 = 'Toggle Blow Off Air'
  1748 = 'Toggle Green Light'
  187 = 'Toggle Pick Up Vauum'
  5 = 'Trigger Camera'
  1782 = 'Tube '
  1108 = 'Tube 1'
  2424 = 'Tube 2'
  1718 = 'Tube 3'
  1340 = 'Tube 4'
  1168 = 'Tube 5'
  1675 = 'Tube Cutting and Inspection System'
  462 = 'Tube Selection '
  989 = 'User Management'
  414 = 'Vacuum'
  2031 = 'vacuum = %0.2f deg/s'
  638 = 'Vacuum = %0.2f mmHg'
  2116 = 'Vacuum Control'
  758 = 'Vacuum Position\t'
  1382 = 'Vacuum Position = %0.2f deg'
  1439 = 'Vacuum Threshold\t'
  1983 = 'Velocities'
  382 = 'Velocity = %0.2f deg/s'
  210 = 'Velocity = %0.2f mm/s'
  591 = 'VelocityX = %0.0f mm/s'
  102 = 'VelocityY = %0.0f mm/s'
  318 = 'View Calibration Info'
  45 = 'View Inspection Results'
  1128 = 'View Raw Data'
  1446 = 'Vision Data and Results (pixels)'
  297 = 'Width = %0.2f px'
  79 = 'x = %0.2f mm'
  311 = 'x = %0.2f mm/s'
  1409 = 'x = %0.3f mm'
  507 = 'x = %0.4f mm'
  1287 = 'X Axis'
  133 = 'X Motor Enable Toggle'
  433 = 'x1 = %0.2f pixel'
  737 = 'x2 = %0.2f pixel'
  290 = 'x3 = %0.2f pixel'
  962 = 'y = %0.2f mm'
  2972 = 'y = %0.2f mm/s'
  1832 = 'y = %0.4f mm'
  661 = 'Y Motor Enable Toggle'
  372 = 'y1 = %0.2f pixel'
  278 = 'y2 = %0.2f pixel'
  1084 = 'y3 = %0.2f pixel'
  266 = 'y= %0.3f mm'
  461 = 'Z Actuator'
END_TEXTLIST

// ---- VISUs/Front_Panel.TcVIS
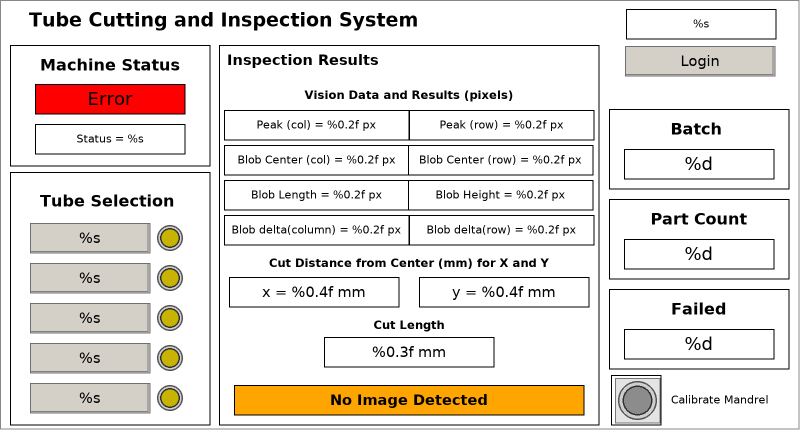
VISUALIZATION Front_Panel  // 800x430
    Rectangle (611,375 50x50), colour toggle: MAIN.fbSlitter.Manual.bCalibrateMandrel
    Frame (214,40 390x390)
        shows Manual_Camera_Inspection()
    Rectangle (10,172 200x253)
    Label (10,186 200x30), "Tube Selection"
    Button (30,223 120x30), "%s", text variable: MAIN.TubeSelection[1].ProductName
        OnMouseClick: execute {
            MAIN.TubeIndicator[1] := TRUE;
            MAIN.TubeIndicator[2] := FALSE;
            MAIN.TubeIndicator[3] := FALSE;
            MAIN.TubeIndicator[4] := FALSE;
            MAIN.TubeIndicator[5] := FALSE;
        }
    Button (30,343 120x30), "%s", text variable: MAIN.TubeSelection[4].ProductName, input disabled if: TRUE
        OnMouseClick: execute {
            MAIN.TubeIndicator[1] := FALSE;
            MAIN.TubeIndicator[2] := FALSE;
            MAIN.TubeIndicator[3] := FALSE;
            MAIN.TubeIndicator[4] := TRUE;
            MAIN.TubeIndicator[5] := FALSE;
        }
    Button (30,383 120x30), "%s", text variable: MAIN.TubeSelection[5].ProductName, input disabled if: TRUE
        OnMouseClick: execute {
            MAIN.TubeIndicator[1] := FALSE;
            MAIN.TubeIndicator[2] := FALSE;
            MAIN.TubeIndicator[3] := FALSE;
            MAIN.TubeIndicator[4] := FALSE;
            MAIN.TubeIndicator[5] := TRUE;
        }
    Lamp1 (155,223 30x30), variable: MAIN.TubeIndicator[1], style: Lamp-Lamp1-Yellow
    Lamp1 (155,263 30x30), variable: MAIN.TubeIndicator[2], style: Lamp-Lamp1-Yellow
    Lamp1 (155,303 30x30), variable: MAIN.TubeIndicator[3], style: Lamp-Lamp1-Yellow
    Lamp1 (155,343 30x30), variable: MAIN.TubeIndicator[4], style: Lamp-Lamp1-Yellow
    Lamp1 (155,383 30x30), variable: MAIN.TubeIndicator[5], style: Lamp-Lamp1-Yellow
    Label (0,5 800x30), "Tube Cutting and Inspection System"
    Rectangle (10,45 200x121)
    Label (10,50 200x30), "Machine Status"
    Rectangle (35,84 150x30), "Initializing", invisible if: MAIN.eState <> E_PMLState.ePMLState_Clearing
    Rectangle (35,84 150x30), "Ready", invisible if: MAIN.eState <> E_PMLState.ePMLState_Idle
    Rectangle (35,84 150x30), "Running", invisible if: MAIN.eState <> E_PMLState.ePMLState_Execute
    Rectangle (35,84 150x30), "Error", invisible if: MAIN.eState <> E_PMLState.ePMLState_Aborted
    Rectangle (609,109 180x80)
    Label (609,114 180x30), "Batch"
    Rectangle (624,149 150x30), "%d", text variable: MAIN.iBatch
        OnMouseClick: write MAIN.hmiBatch via Default, title 'Batch Number'
    Rectangle (609,199 180x80)
    Label (609,204 180x30), "Part Count"
    Rectangle (624,239 150x30), "%d", text variable: MAIN.iCounter
    Rectangle (609,289 180x80)
    Label (609,294 180x30), "Failed"
    Rectangle (624,329 150x30), "%d", text variable: MAIN.iCountFailed
    Rectangle (35,124 150x30), "Status = %s", text variable: MAIN.hmiStatus
    Rectangle (626,9 150x30), "%s", text variable: MAIN.currentUser
    Button (625,46 150x30), "Login"
        OnMouseClick: VisuUserMgmt Type=Login
    PushSwitch (615,378 45x45), variable: MAIN.fbSlitter.Manual.bCalibrateMandrel, behaviour: TOGGLE, style: Switch-PushSwitch-Gray
    Label (668,385 111x30), "Calibrate Mandrel"
    Button (30,263 120x30), "%s", text variable: MAIN.TubeSelection[2].ProductName
        OnMouseClick: execute {
            MAIN.TubeIndicator[1] := FALSE;
            MAIN.TubeIndicator[2] := TRUE;
            MAIN.TubeIndicator[3] := FALSE;
            MAIN.TubeIndicator[4] := FALSE;
            MAIN.TubeIndicator[5] := FALSE;
        }
    Button (30,303 120x30), "%s", text variable: MAIN.TubeSelection[3].ProductName
        OnMouseClick: execute {
            MAIN.TubeIndicator[1] := FALSE;
            MAIN.TubeIndicator[2] := FALSE;
            MAIN.TubeIndicator[3] := TRUE;
            MAIN.TubeIndicator[4] := FALSE;
            MAIN.TubeIndicator[5] := FALSE;
        }
END_VISUALIZATION

// ---- VISUs/Manual_Inspect.TcVIS
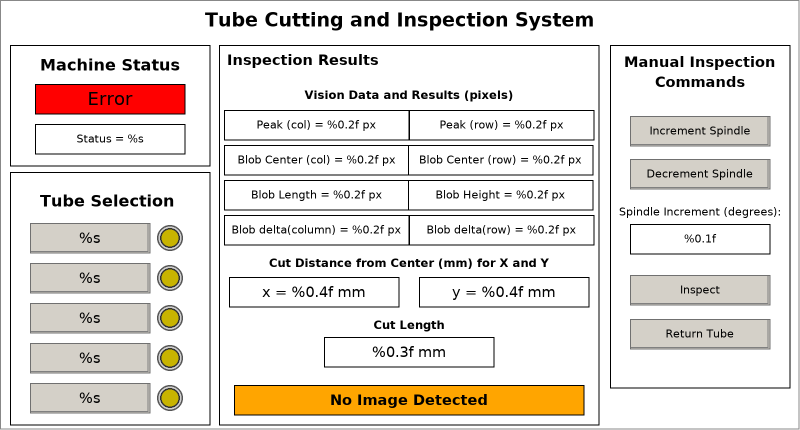
VISUALIZATION Manual_Inspect  // 800x430
    Rectangle (610,45 180x343)
    Frame (214,40 390x390)
        shows Manual_Camera_Inspection()
    Rectangle (10,172 200x253)
    Label (10,186 200x30), "Tube Selection"
    Button (30,223 120x30), "%s", text variable: MAIN.TubeSelection[1].ProductName
        OnMouseClick: execute {
            MAIN.TubeIndicator[1] := TRUE;
            MAIN.TubeIndicator[2] := FALSE;
            MAIN.TubeIndicator[3] := FALSE;
            MAIN.TubeIndicator[4] := FALSE;
            MAIN.TubeIndicator[5] := FALSE;
        }
    Button (30,263 120x30), "%s", text variable: MAIN.TubeSelection[2].ProductName
        OnMouseClick: execute {
            MAIN.TubeIndicator[1] := FALSE;
            MAIN.TubeIndicator[2] := TRUE;
            MAIN.TubeIndicator[3] := FALSE;
            MAIN.TubeIndicator[4] := FALSE;
            MAIN.TubeIndicator[5] := FALSE;
        }
    Button (30,303 120x30), "%s", text variable: MAIN.TubeSelection[3].ProductName
        OnMouseClick: execute {
            MAIN.TubeIndicator[1] := FALSE;
            MAIN.TubeIndicator[2] := FALSE;
            MAIN.TubeIndicator[3] := TRUE;
            MAIN.TubeIndicator[4] := FALSE;
            MAIN.TubeIndicator[5] := FALSE;
        }
    Button (30,343 120x30), "%s", text variable: MAIN.TubeSelection[4].ProductName, input disabled if: TRUE
        OnMouseClick: execute {
            MAIN.TubeIndicator[1] := FALSE;
            MAIN.TubeIndicator[2] := FALSE;
            MAIN.TubeIndicator[3] := FALSE;
            MAIN.TubeIndicator[4] := TRUE;
            MAIN.TubeIndicator[5] := FALSE;
        }
    Button (30,383 120x30), "%s", text variable: MAIN.TubeSelection[5].ProductName, input disabled if: TRUE
        OnMouseClick: execute {
            MAIN.TubeIndicator[1] := FALSE;
            MAIN.TubeIndicator[2] := FALSE;
            MAIN.TubeIndicator[3] := FALSE;
            MAIN.TubeIndicator[4] := FALSE;
            MAIN.TubeIndicator[5] := TRUE;
        }
    Lamp1 (155,223 30x30), variable: MAIN.TubeIndicator[1], style: Lamp-Lamp1-Yellow
    Lamp1 (155,263 30x30), variable: MAIN.TubeIndicator[2], style: Lamp-Lamp1-Yellow
    Lamp1 (155,303 30x30), variable: MAIN.TubeIndicator[3], style: Lamp-Lamp1-Yellow
    Lamp1 (155,343 30x30), variable: MAIN.TubeIndicator[4], style: Lamp-Lamp1-Yellow
    Lamp1 (155,383 30x30), variable: MAIN.TubeIndicator[5], style: Lamp-Lamp1-Yellow
    Label (0,5 800x30), "Tube Cutting and Inspection System"
    Rectangle (10,45 200x121)
    Label (10,50 200x30), "Machine Status"
    Rectangle (35,84 150x30), "Initializing", invisible if: MAIN.eState <> E_PMLState.ePMLState_Clearing
    Rectangle (35,84 150x30), "Ready", invisible if: MAIN.eState <> E_PMLState.ePMLState_Idle
    Rectangle (35,84 150x30), "Running", invisible if: MAIN.eState <> E_PMLState.ePMLState_Execute
    Rectangle (35,84 150x30), "Error", invisible if: MAIN.eState <> E_PMLState.ePMLState_Aborted
    Rectangle (35,124 150x30), "Status = %s", text variable: MAIN.hmiStatus
    Button (630,116 140x30), "Increment Spindle"
        tap MAIN.InspectCommands.IncrementSpindle
        OnMouseClick: execute { MAIN.fbSlitter.bIncrementSpindle := TRUE; }
    Button (630,275 140x30), "Inspect"
        tap MAIN.InspectCommands.Inspect
        OnMouseClick: execute { MAIN.fbSlitter.bInspect := TRUE; }
    Label (610,47 180x30), "Manual Inspection"
    Label (610,67 180x30), "Commands"
    Button (630,159 140x30), "Decrement Spindle"
        tap MAIN.InspectCommands.DecrementSpindle
        OnMouseClick: execute { MAIN.fbSlitter.bDecrementSpindle := TRUE; }
    Button (630,319 140x30), "Return Tube"
        tap MAIN.InspectCommands.InspectComplete
        OnMouseClick: execute { MAIN.fbSlitter.bInspectComplete := TRUE; }
    Rectangle (630,224 140x30), "%0.1f", text variable: MAIN.fbSlitter.Mandrel._SpindleIncrement
        OnMouseClick: write MAIN.fbSlitter.Mandrel._SpindleIncrement via Default
    Label (620,197 160x30), "Spindle Increment (degrees):"
END_VISUALIZATION

// ---- VISUs/MachineSettings.TcVIS
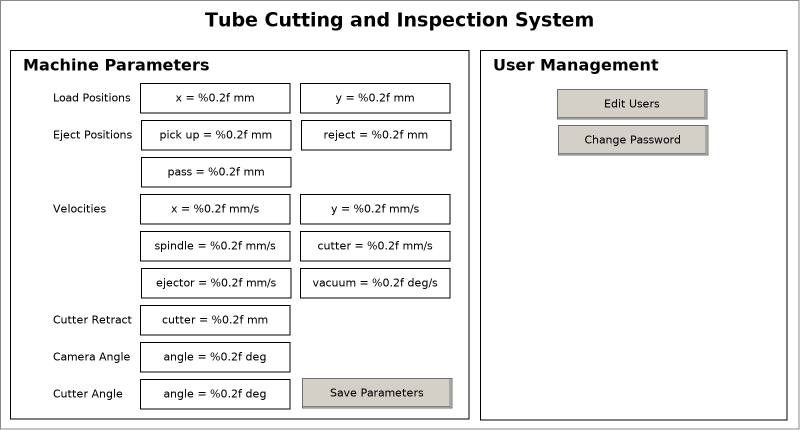
VISUALIZATION MachineSettings  // 800x430
    Label (0,5 800x30), "Tube Cutting and Inspection System"
    Rectangle (10,50 459x369)
    Button (302,378 150x30), "Save Parameters"
        OnMouseClick: execute { MAIN.bSave := TRUE; }
    Label (50,83 90x30), "Load Positions"
    Rectangle (140,83 150x30), "x = %0.2f mm", text variable: MAIN.fbSlitter.Mandrel._hmiParameters.loadPositionX
        OnMouseClick: write MAIN.fbSlitter.Mandrel._hmiParameters.loadPositionX via Default, title 'Load Position X'
    Rectangle (300,83 150x30), "y = %0.2f mm", text variable: MAIN.fbSlitter.Mandrel._hmiParameters.loadPositionY
        OnMouseClick: write MAIN.fbSlitter.Mandrel._hmiParameters.loadPositionY via Default, title 'Load Position Y'
    Label (50,194 90x30), "Velocities"
    Rectangle (140,194 150x30), "x = %0.2f mm/s", text variable: MAIN.fbSlitter.Mandrel._hmiParameters.velocityX
        OnMouseClick: write MAIN.fbSlitter.Mandrel._hmiParameters.VelocityX via Default, title 'X Axis Velocity'
    Rectangle (300,194 150x30), "y = %0.2f mm/s", text variable: MAIN.fbSlitter.Mandrel._hmiParameters.velocityY
        OnMouseClick: write MAIN.fbSlitter.Mandrel._hmiParameters.velocityY via Default, title 'Y Axis Velocity'
    Rectangle (140,231 150x30), "spindle = %0.2f mm/s", text variable: MAIN.fbSlitter.Mandrel._hmiParameters.spindleVelocity
        OnMouseClick: write MAIN.fbSlitter.Mandrel._hmiParameters.spindleVelocity via Default, title 'Spindle Velocity'
    Rectangle (300,231 150x30), "cutter = %0.2f mm/s", text variable: MAIN.fbSlitter.Cutter._hmiParameters.cutVelocity
        OnMouseClick: write MAIN.fbSlitter.Cutter._hmiParameters.cutVelocity via Default, title 'Cutter Axis Velocity'
    Label (50,305 90x30), "Cutter Retract"
    Rectangle (140,305 150x30), "cutter = %0.2f mm", text variable: MAIN.fbSlitter.Cutter._hmiParameters.retractPosition
        OnMouseClick: write MAIN.fbSlitter.Cutter._hmiParameters.retractPosition via Default, title 'Cutter Retract Position'
    Rectangle (140,342 150x30), "angle = %0.2f deg", text variable: MAIN.fbSlitter.Camera._hmiParameters.angle
        OnMouseClick: write MAIN.fbSlitter.Camera._hmiParameters.angle via Default, title 'Camera Angle'
    Label (50,342 90x30), "Camera Angle"
    Label (20,50 189x30), "Machine Parameters"
    Rectangle (140,379 150x30), "angle = %0.2f deg", text variable: MAIN.fbSlitter.Mandrel._hmiParameters.spindleOffset
        OnMouseClick: write MAIN.fbSlitter.Mandrel._hmiParameters.spindleOffset via Default, title 'Cutter to Camera Angular Offset'
    Label (50,379 90x30), "Cutter Angle"
    Rectangle (480,50 307x370)
    Label (490,50 189x30), "User Management"
    Button (557,89 150x30), "Edit Users"
        OnMouseClick: VisuUserMgmt Type=OpenUserConfiguration
    Button (558,125 150x30), "Change Password"
        OnMouseClick: VisuUserMgmt Type=ChangeUserPassword
    Rectangle (141,268 150x30), "ejector = %0.2f mm/s", text variable: MAIN.fbSlitter.Ejector._hmiParameters.ejectVelocity
        OnMouseClick: write MAIN.fbSlitter.Ejector._hmiParameters.ejectVelocity via Default, title 'Ejector Axis Velocity'
    Label (50,120 90x30), "Eject Positions"
    Rectangle (141,120 150x30), "pick up = %0.2f mm", text variable: MAIN.fbSlitter.Ejector._hmiParameters.ejectPositionHome
        OnMouseClick: write MAIN.fbSlitter.Ejector._hmiParameters.ejectPositionHome via Default, title 'Eject Pick Up Position'
    Rectangle (301,120 150x30), "reject = %0.2f mm", text variable: MAIN.fbSlitter.Ejector._hmiParameters.ejectPositionFail
        OnMouseClick: write MAIN.fbSlitter.Ejector._hmiParameters.ejectPositionFail via Default, title 'Reject Position'
    Rectangle (141,157 150x30), "pass = %0.2f mm", text variable: MAIN.fbSlitter.Ejector._hmiParameters.ejectPositionPass
        OnMouseClick: write MAIN.fbSlitter.Ejector._hmiParameters.ejectPositionPass via Default, title 'Eject Pass Position'
    Rectangle (300,268 150x30), "vacuum = %0.2f deg/s", text variable: MAIN.fbSlitter.Mandrel._hmiParameters.vacuumVelocity
        OnMouseClick: write MAIN.fbSlitter.Mandrel._hmiParameters.vacuumVelocity via Default, min 0, max 360, title 'Vacuum Axis Velocity'
END_VISUALIZATION

// ---- VISUs/ManualControl.TcVIS
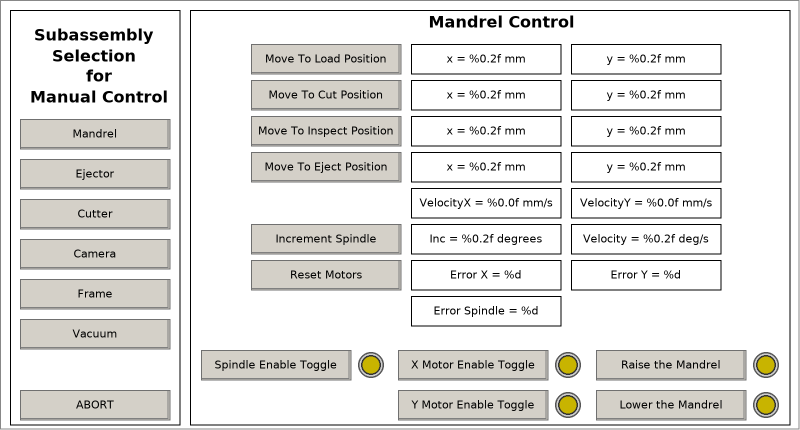
VISUALIZATION ManualControl  // 800x430
    Rectangle (190,10 600x415)
    Frame (191,0 600x430)
        shows Manual_Mandrel()
        shows Manual_Ejector()
        shows Manual_Cutter()
        shows Manual_Camera()
        shows Manual_Frame()
        shows Manual_Select_Tube()
        shows Manual_Vacuum()
    Rectangle (10,10 170x415)
    Button (20,119 150x30), "Mandrel"
        OnMouseClick: FrameSelectionChange Selection=SelectedFrame=b6e51242-079a-4729-85ea-e161656839df, GlobSel=AssignType=Directly, SelType=Locally
        OnMouseClick: execute { MAIN.TubeHmi := Main.Tube; }
    Button (20,159 150x30), "Ejector"
        OnMouseClick: FrameSelectionChange Selection=SelectedFrame=b6e51242-079a-4729-85ea-e161656839df, Selection=1, GlobSel=AssignType=Directly, SelType=Locally
    Button (20,199 150x30), "Cutter"
        OnMouseClick: FrameSelectionChange Selection=SelectedFrame=b6e51242-079a-4729-85ea-e161656839df, Selection=2, GlobSel=AssignType=Directly, SelType=Locally
    Button (20,239 150x30), "Camera"
        OnMouseClick: FrameSelectionChange Selection=SelectedFrame=b6e51242-079a-4729-85ea-e161656839df, Selection=3, GlobSel=AssignType=Directly, SelType=Locally
    Button (20,279 150x30), "Frame"
        OnMouseClick: FrameSelectionChange Selection=SelectedFrame=b6e51242-079a-4729-85ea-e161656839df, Selection=4, GlobSel=AssignType=Directly, SelType=Locally
    Button (20,390 150x30), "ABORT"
        OnMouseClick: execute { MAIN.eCommand := E_PMLCommand.ePMLCommand_Abort; }
    Group (10,20 170x92)
        Group (0,0 170x51)
            Label (0,21 168x30), "Selection"
            Label (0,0 168x30), "Subassembly"
        Label (4,62 170x30), "Manual Control"
        Label (4,41 170x30), "for"
    Button (20,319 150x30), "Vacuum"
        OnMouseClick: FrameSelectionChange Selection=SelectedFrame=b6e51242-079a-4729-85ea-e161656839df, Selection=6, GlobSel=AssignType=Directly, SelType=Locally
END_VISUALIZATION

// ---- VISUs/Manual_Camera.TcVIS
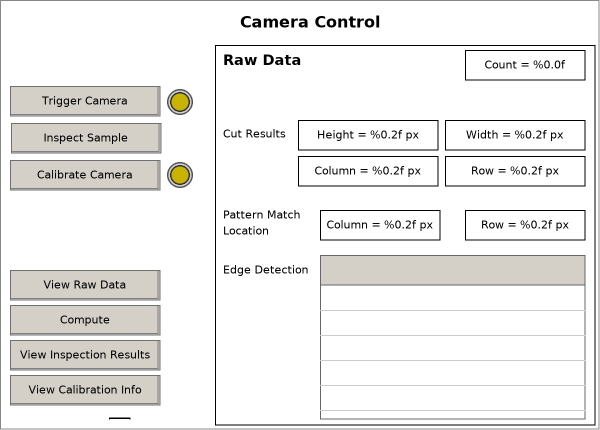
VISUALIZATION Manual_Camera  // 600x430
    Label (133,7 355x30), "Camera Control"
    Button (11,123 150x30), "Inspect Sample", input disabled if: MAIN.fbSlitter.bBusy
        OnMouseClick: execute { MAIN.fbSlitter.Manual.bCameraInspect := TRUE; }
    Button (10,86 150x30), "Trigger Camera", input disabled if: MAIN.fbSlitter.bBusy
        OnMouseClick: execute { MAIN.fbSlitter.Manual.bCameraTrigger := TRUE; }
    Button (10,160 150x30), "Calibrate Camera", input disabled if: MAIN.fbSlitter.bBusy
        OnMouseClick: execute { MAIN.fbSlitter.Manual.bCameraCalibrate := TRUE; }
        OnMouseClick: FrameSelectionChange Selection=SelectedFrame=62eee777-8d81-454f-aaa1-e694c65750cd, Selection=2, GlobSel=AssignType=Directly, SelType=Locally
    Lamp1 (165,87 30x30), variable: MAIN.fbSlitter.Camera.Trigger, style: Lamp-Lamp1-Yellow
    Lamp1 (165,160 30x30), variable: MAIN.fbSlitter.bCalibration, style: Lamp-Lamp1-Yellow
    Frame (210,40 390x390)
        shows Manual_Camera_RawData()
        shows Manual_Camera_Inspection_Raw()
        shows Manual_Camera_Calibration()
        shows Manual_Select_Tube()
    Button (10,270 150x30), "View Raw Data"
        OnMouseClick: FrameSelectionChange Selection=SelectedFrame=62eee777-8d81-454f-aaa1-e694c65750cd, GlobSel=AssignType=Directly, SelType=Locally
        OnMouseClick: execute { MAIN.fbSlitter.Manual.bCameraRawData := TRUE; }
    Button (10,340 150x30), "View Inspection Results"
        OnMouseClick: FrameSelectionChange Selection=SelectedFrame=62eee777-8d81-454f-aaa1-e694c65750cd, Selection=1, GlobSel=AssignType=Directly, SelType=Locally
    Button (10,375 150x30), "View Calibration Info"
        OnMouseClick: FrameSelectionChange Selection=SelectedFrame=62eee777-8d81-454f-aaa1-e694c65750cd, Selection=2, GlobSel=AssignType=Directly, SelType=Locally
    Button (10,305 150x30), "Compute"
        OnMouseClick: execute { Main.fbSlitter.Manual.bCameraComputePeak := TRUE; }
    Rectangle (109,418 21x0)
END_VISUALIZATION

// ---- VISUs/Manual_Camera_Calibration.TcVIS
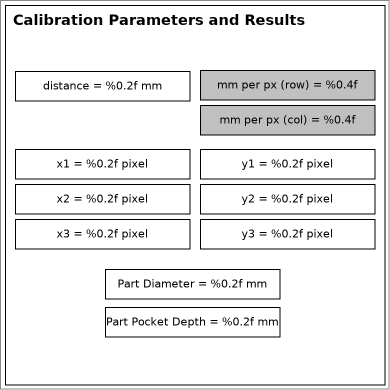
VISUALIZATION Manual_Camera_Calibration  // 390x390
    Rectangle (5,5 380x380)
    Rectangle (15,149 175x30), "x1 = %0.2f pixel", text variable: MAIN.fbSlitter.Camera._patternX1
    Rectangle (200,149 175x30), "y1 = %0.2f pixel", text variable: MAIN.fbSlitter.Camera._patternY1
    Rectangle (15,184 175x30), "x2 = %0.2f pixel", text variable: MAIN.fbSlitter.Camera._patternX2
    Rectangle (200,184 175x30), "y2 = %0.2f pixel", text variable: MAIN.fbSlitter.Camera._patternY2
    Rectangle (15,71 175x30), "distance = %0.2f mm", text variable: MAIN.fbSlitter.Camera._hmiParameters.calibrationDistance
        OnMouseClick: write MAIN.fbSlitter.Camera._hmiParameters.calibrationDistance via Default, title 'Load Position X'
    Rectangle (200,70 175x30), "mm per px (row) = %0.4f", text variable: MAIN.fbSlitter.Camera._parameters.pitchRow
    Label (10,5 297x30), "Calibration Parameters and Results"
    Rectangle (105,269 175x30), "Part Diameter = %0.2f mm", text variable: MAIN.fbSlitter.Camera._tubeParameters.Diameter
    Rectangle (105,307 175x30), "Part Pocket Depth = %0.2f mm", text variable: MAIN.fbSlitter.Camera._tubeParameters.DepthOfPocket
    Rectangle (15,219 175x30), "x3 = %0.2f pixel", text variable: MAIN.fbSlitter.Camera._patternX3
    Rectangle (200,219 175x30), "y3 = %0.2f pixel", text variable: MAIN.fbSlitter.Camera._patternY3
    Rectangle (200,105 175x30), "mm per px (col) = %0.4f", text variable: MAIN.fbSlitter.Camera._parameters.pitchColumn
END_VISUALIZATION

// ---- VISUs/Manual_Camera_Inspection.TcVIS
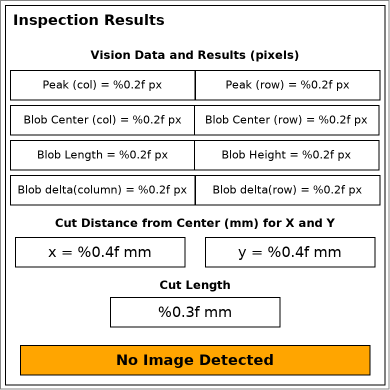
VISUALIZATION Manual_Camera_Inspection  // 390x390
    Rectangle (5,5 380x380)
    Rectangle (20,345 350x30), "PASSED", invisible if: NOT MAIN.bPassed
    Rectangle (20,345 350x30), "FAILED", invisible if: NOT MAIN.bFailed
    Rectangle (20,345 350x30), "Processing", invisible if: NOT MAIN.bProcessing
    Label (10,5 297x30), "Inspection Results"
    Rectangle (10,70 185x30), "Peak (col) = %0.2f px", text variable: MAIN.fbSlitter.Camera._columnPeak
    Rectangle (195,70 185x30), "Peak (row) = %0.2f px", text variable: MAIN.fbSlitter.Camera._rowPeak
    Rectangle (10,105 185x30), "Blob Center (col) = %0.2f px", text variable: MAIN.fbSlitter.Camera.CameraData.Results.LocationInX
    Rectangle (194,105 185x30), "Blob Center (row) = %0.2f px", text variable: MAIN.fbSlitter.Camera.CameraData.Results.LocationInY
    Rectangle (10,175 185x30), "Blob delta(column) = %0.2f px", text variable: MAIN.fbSlitter.Camera.DeltaXpx
    Rectangle (195,175 185x30), "Blob delta(row) = %0.2f px", text variable: MAIN.fbSlitter.Camera.DeltaYpx
    Rectangle (15,237 170x30), "x = %0.4f mm", text variable: MAIN.fbSlitter.Camera._DeltaXmmWithOffset
    Rectangle (205,237 170x30), "y = %0.4f mm", text variable: MAIN.fbSlitter.Camera._DeltaYmmWithOffset
    Label (0,208 390x30), "Cut Distance from Center (mm) for X and Y"
    Rectangle (110,297 170x30), "%0.3f mm", text variable: MAIN.fbSlitter.Camera._CutLengthWithOffset
    Label (0,40 390x30), "Vision Data and Results (pixels)"
    Rectangle (10,140 185x30), "Blob Length = %0.2f px", text variable: MAIN.fbSlitter.Camera.CameraData.Results.WidthMeasurement
    Rectangle (194,140 185x30), "Blob Height = %0.2f px", text variable: MAIN.fbSlitter.Camera.CameraData.Results.HeightMeasurement
    Label (0,270 390x30), "Cut Length"
    Rectangle (20,345 350x30), "No Image Detected", invisible if: NOT MAIN.bNoDetect
END_VISUALIZATION

// ---- VISUs/Manual_Camera_Inspection_Raw.TcVIS
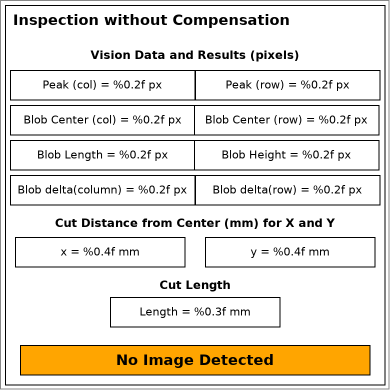
VISUALIZATION Manual_Camera_Inspection_Raw  // 390x390
    Rectangle (20,345 350x30), "PASSED", invisible if: NOT MAIN.bPassed
    Rectangle (20,345 350x30), "FAILED", invisible if: NOT MAIN.bFailed
    Rectangle (5,5 380x380)
    Label (10,5 297x30), "Inspection without Compensation"
    Rectangle (10,70 185x30), "Peak (col) = %0.2f px", text variable: MAIN.fbSlitter.Camera._columnPeak
    Rectangle (195,70 185x30), "Peak (row) = %0.2f px", text variable: MAIN.fbSlitter.Camera._rowPeak
    Rectangle (10,105 185x30), "Blob Center (col) = %0.2f px", text variable: MAIN.fbSlitter.Camera.CameraData.Results.LocationInX
    Rectangle (194,105 185x30), "Blob Center (row) = %0.2f px", text variable: MAIN.fbSlitter.Camera.CameraData.Results.LocationInY
    Rectangle (10,175 185x30), "Blob delta(column) = %0.2f px", text variable: MAIN.fbSlitter.Camera.DeltaXpx
    Rectangle (195,175 185x30), "Blob delta(row) = %0.2f px", text variable: MAIN.fbSlitter.Camera.DeltaYpx
    Rectangle (15,237 170x30), "x = %0.4f mm", text variable: MAIN.fbSlitter.Camera.DeltaXmm
    Rectangle (205,237 170x30), "y = %0.4f mm", text variable: MAIN.fbSlitter.Camera.DeltaYmm
    Label (0,208 390x30), "Cut Distance from Center (mm) for X and Y"
    Rectangle (110,297 170x30), "Length = %0.3f mm", text variable: MAIN.fbSlitter.Camera.CutLength
    Label (0,40 390x30), "Vision Data and Results (pixels)"
    Rectangle (10,140 185x30), "Blob Length = %0.2f px", text variable: MAIN.fbSlitter.Camera.CameraData.Results.WidthMeasurement
    Rectangle (194,140 185x30), "Blob Height = %0.2f px", text variable: MAIN.fbSlitter.Camera.CameraData.Results.HeightMeasurement
    Label (0,270 390x30), "Cut Length"
    Rectangle (20,345 350x30), "Processing", invisible if: NOT MAIN.bProcessing
    Rectangle (20,345 350x30), "No Image Detected", invisible if: NOT MAIN.bNoDetect
END_VISUALIZATION

